(* IEC 61131-3 sources: Mizera_Tube/Plc (part 10) *)

LD   xEnFIR                        ** Abilita filtri FIR
ST   StPrFilterEnab                ** Stato precedente abilitazione filtri

LDN  xEnFIR                        ** Abilita filtri FIR
ST   EFCR_NF_DISABLE               ** NanoFIR subsystem disable

LDN  xEnFIR                        ** Abilita filtri FIR
ORN  EFSR_ACK_NF_DISABLE           ** ACK nanoFIR subsystem disable
AND  (
LD   xEnFIR                        ** Abilita filtri FIR
OR   EFSR_ACK_NF_DISABLE           ** ACK nanoFIR subsystem disable
)
ST   EFCR_SUBSYSTEM_EN             ** Filter subsystem master enable

LD   yLimiter                      ** Intervento limitatore
OR   xSetAlarm                     ** Forzamento allarme asse
*ANDN %ra0.28       ** Mem. collegamento richiesto con albero elettrico
ST   BAI_SETALARM                  ** ra0.27 Richiesta allarme asse

LD   xUnlock                       * reset gestax
R    yLimiter                      ** Intervento limitatore

LD   xEnFrComp                     ** Abilita friction compensation
ST   EFCR_FRICTION_COMP            ** Enable static friction comp.
ST   EFCR_RT_CHANGES_EN            ** Enable run-time changes (RT)

* Alarm if there is request of closeloop without drive enable

LD   BAI_CHAN                      ** ra0.0 Chiusura anello di posizione
AND  (
LD   %nvel11
EQ   3
OR   (
LD   %nvel11
EQ   4
)
)
ANDN BAI_AXEN                      ** Drive is enabled
ANDN LINK_SIMUL                    ** PLCFLAGS.16 LINK=SIMUL
ANDN AP_OPZIONI31                  ** pa3.31 Asse in simulato
ST   alarmEn                       ** Drive is disable, with enable request enabled

CAL  TON_ALARM_DISABLE (IN:=alarmEn,PT:=2000) ** Drive is disable, with enable request enabled

LD   TON_ALARM_DISABLE.Q
ST   yDriveNotEn                   ** Closeloop but drive not enabled (alarm)

LD  TON_ALARM_DISABLE.Q
JMPCN drive_is_enabled

LD   ALWAYS_ZERO                   ** PLCFLAGS.0  Flag sempre stato off
ST   AX_DRV_ENAB                   ** rg0.13 signal to understand all drives are enabled
drive_is_enabled:

* Comando bit avanti e indietro per i modi REF, JOG, INC

LD   CMD_START_AXIS                ** rgc0.5 Comando start assi canale
ANDN xLockRef                      ** Blocco avvio ciclo REF da canale
OR   xEnabRef                      ** Abilita avvio ciclo REF
AND  BCI_TAR                       ** rc0.8  Selettore modi operativi su REF (taratura)
AND  (
LDN  xZeroForced                   ** Forzamento asse tarato
ANDN BSC_SINGREF                   ** rgc0.18 Selezione modo REF singolo nel canale
OR   (
LD   xSelected                     ** Asse selezionato
AND  BSC_SINGREF                   ** rgc0.18 Selezione modo REF singolo nel canale
)
)
ST   StartRef                      ** Avvio ciclo di taratura

LD   CMD_PLUS_AXIS                 ** rgc0.0 Comando + assi canale
AND  xSelected                     ** Asse selezionato
OR   xJogPlus                      ** Comando manuale avanti
AND  AX_EXEC_MODE                  ** rgc0.3 Canale in JOG o INC
OR(
LD   StartRef                      ** Avvio ciclo di taratura
AND  AP_OPZIONI0                   ** pa3.0 Bit inversione direzione taratura
ANDN AsseNvel                      ** Asse di tipo NVEL
)
OR(
LD   StartRef                      ** Avvio ciclo di taratura
AND  NV_OPZIONI0                   ** pa1.0 Bit inversione direzione taratura (NVEL)
AND  AsseNvel                      ** Asse di tipo NVEL
)
ST   BAI_AV                        ** ra0.8 Comando avanti

LD   CMD_MINUS_AXIS                ** rgc0.1 Comando - assi canale
AND  xSelected                     ** Asse selezionato
OR   xJogMinus                     ** Comando manuale indietro
AND  AX_EXEC_MODE                  ** rgc0.3 Canale in JOG o INC
OR(
LD   StartRef                      ** Avvio ciclo di taratura
ANDN AP_OPZIONI0                   ** pa3.0 Bit inversione direzione taratura
ANDN AsseNvel                      ** Asse di tipo NVEL
)
OR(
LD   StartRef                      ** Avvio ciclo di taratura
ANDN NV_OPZIONI0                   ** pa1.0 Bit inversione direzione taratura (NVEL)
AND  AsseNvel                      ** Asse di tipo NVEL
)
ST   BAI_IND                       ** ra0.9 Comando indietro

* Passaggio finecorsa taratura e limite

LD   xRefLS                        ** Finecorsa di taratura
ST   BAI_FCRALL                    ** ra0.13 Finecorsa Taratura

LD   xPlusLS                       ** Finecorsa +
ST   BAI_FCHWAV                    ** ra0.10 Finecorsa avanti

LD   xMinusLS                      ** Finecorsa -
ST   BAI_FCHWIN                    ** ra0.11 Finecorsa indietro

* Reset asse in allarme

LD   CMD_RESET_AXIS                ** rgc0.4 Comando reset assi canale
ST   BAI_RESALARM                  ** ra0.15 Ripristino allarme asse

* Full-handshake motion block sul singolo asse

LD   BAO_STB_PLC_SYNC              ** ra22.16 strobe Full-handshake Motion block asse
AND  ACK_AX_FHMB                   ** rgc0.8 Abil. ACK Full-handshake Motion block per assi
ST   BAI_ACK_PLC_SYNC              ** ra0.26 ACK Full-handshake Motion block asse

* Taratura immediata (preset) sul singolo asse

LD   BSC_PRESETREF                 ** rgc0.19 Selezione modo REF preset nel canale
ST   BAI_TARAIM                    ** ra0.24 Selezione taratura immediata

LD   SC_QTAIMM                     ** rgc6 Quota per taratura immediata (preset)
ST   AI_QTAIMM                     ** ra2  Quota taratura immediata

* JOG DA VOLANTINO

LD   xSelected                     ** Asse selezionato
AND  PA_MOV_JOG                    ** rg0.8 Richiesta movim. da volantino in JOG
ST   JOG_AX.xax_ENABLE

LDN  JOG_AX.xax_ENABLE
ST   JOG_AX.xax_CLEAR

LD   JOG_AX.xax_ENABLE
AND  JOG_AX.yax_READY
ANDN JOG_AX.yax_RUNNING
AND  (
LDN  JOG_AX.yax_ENDERR
OR   JOG_AX.yax_ERRCODE.1
)
ST   JOG_AX.xax_START

LDN  PA_INV_DIR                    ** rg0.7 Movim. da volantino in direzione inversa
ST   JOG_AX.xax_REVERSE

CAL  JOG_AX

* Rileva il cambio di selezione asse

CAL  RT_AXSEL(CLK=xSelected)       ** Asse selezionato

LD   RT_AXSEL.Q                    ** Imp. selezione asse
S    AX_SEL_CHG                    ** rg0.12 Imp. modifica selezione asse

* POSIZIONAMENTO TRAMITE VOLANTINO

LD   xSelected                     ** Asse selezionato
ANDN RT_AXSEL.Q                    ** Imp. selezione asse
AND  PA_ENAB_POS                   ** rg0.9 Abilita posiz. asse da volantino
ST   POS_AX.xax_ENABLE

LDN  POS_AX.xax_ENABLE
ST   POS_AX.xax_CLEAR

LD   SG_QTAR_PAUX                  ** rg9 Quota Target per posiz. da puls. aux
NE   AO_QUOTA                      ** ra4  Quota asse
AND  POS_AX.xax_ENABLE
AND  POS_AX.yax_READY
ANDN POS_AX.yax_RUNNING
ANDN POS_AX.yax_ENDERR
ST   POS_AX.xax_START

LD   SG_QTAR_PAUX                  ** rg9 Quota Target per posiz. da puls. aux
ST   POS_AX.xax_QUOTA

LD   SG_VEL_PAUX                   ** rg14 Velocit� per posiz. da puls. aux
ST   POS_AX.xax_VEL

LD   SG_VEL_PAUX                   ** rg14 Velocit� per posiz. da puls. aux
GT   AP_VELMAX                     ** pa9 Velocit� massima
JMPCN END_VMAX

LD   AP_VELMAX                     ** pa9 Velocit� massima
ST   POS_AX.xax_VEL

END_VMAX:

CAL  POS_AX

* ALBERO ELETTRICO (per volantino e G4010)

LD   xSelected                     ** Asse selezionato
AND  PA_ENAB_ELS                   ** rg0.11 Abilita albero elettrico da volantino
OR   MemConnAE                     ** Mem. collegamento richiesto con albero elettrico
ANDN CAM_AX.yax_RUNNING
ST   EL_SH.xax_ENABLE

LDN  EL_SH.xax_ENABLE
OR   EL_SH.yax_ENDERR
ST   EL_SH.xax_CLEAR

LD   EL_SH.xax_ENABLE
AND  EL_SH.yax_READY
ANDN EL_SH.yax_ENDOK
ANDN EL_SH.yax_ENDERR
ANDN EL_SH.yax_RUNNING
ST   EL_SH.xax_START

LD   MemConnAE                     ** Mem. collegamento richiesto con albero elettrico
JMPC ELS_CON

LD   PA_INCJOG                     ** QPuls2 Quota incremento per posiz. da volantino
ST   EL_SH.xax_TRNUM

LD   EL_SH.xax_TRNUM
LT   1
JMPCN END_TRLIM

LD   1
ST   EL_SH.xax_TRNUM

END_TRLIM:

LD   1
ST   EL_SH.xax_TRDEN

LD   128
ST   EL_SH.xax_MODE

LD   SG_VOLAX                      ** rg16 Numero asse master per volantino
ST   EL_SH.xax_MASTER

JMP  ELS_END

ELS_CON:

LD   1
ST   EL_SH.xax_TRNUM
ST   EL_SH.xax_TRDEN

LD   0
ST   EL_SH.xax_MODE

LD   CONN_MAST                     ** rga1 Numero asse master per aggancio albero elettrico
ST   EL_SH.xax_MASTER

ELS_END:

CAL  EL_SH

* AX COUPLING

LD   MemConnCP                     ** Mem. collegamento richiesto con coupling
ANDN EL_SH.yax_RUNNING
ST   CAM_AX.xax_ENABLE

LDN  CAM_AX.xax_ENABLE
ST   CAM_AX.xax_CLEAR

LD   CAM_AX.xax_ENABLE
AND  CAM_AX.yax_READY
ANDN CAM_AX.yax_ENDOK
ANDN CAM_AX.yax_ENDERR
ST   CAM_AX.xax_START

LD   CP_TYPEC                      ** rga7 Tipo connessione per coupling
ST   CAM_AX.xax_MODE

*LD   0                      *non disponibile*
*ST   CAM_AX.xax_INSTANCE

LD   CP_MAST1                      ** rga3 Numero asse master 1 per coupling
ST   CAM_AX.xax_MASTER0

LD   CP_MAST2                      ** rga4 Numero asse master 2 per coupling
ST   CAM_AX.xax_MASTER1

LD   CP_MAST3                      ** rga5 Numero asse master 3 per coupling
ST   CAM_AX.xax_MASTER2

LD   CP_MAST4                      ** rga6 Numero asse master 4 per coupling
ST   CAM_AX.xax_MASTER3

LD   -1
ST   CAM_AX.xax_MASTER4

LD   -1
ST   CAM_AX.xax_MASTER5

CAL  CAM_AX

* Conferma comando effettuato

LD   MemConnAE                     ** Mem. collegamento richiesto con albero elettrico
AND  EL_SH.yax_RUNNING
AND  %ra8.14             * Conferma albero elettrico agganciato
OR   BAO_ALLM                      ** ra3.15  Asse in Allarme
OR   BAI_RESALARM                  ** ra0.15 Ripristino allarme asse
AND  REQ_CONN_AX                   ** rga0.0 Richiesta aggancio asse in albero elettrico
R    REQ_CONN_AX                   ** rga0.0 Richiesta aggancio asse in albero elettrico

LD   MemConnCP                     ** Mem. collegamento richiesto con coupling
AND  CAM_AX.yax_RUNNING
AND  %ra8.14             * Conferma albero elettrico agganciato
OR   BAO_ALLM                      ** ra3.15  Asse in Allarme
OR   BAI_RESALARM                  ** ra0.15 Ripristino allarme asse
AND  REQ_CONN_CP                   ** rga0.2 Richiesta aggancio asse in coupling
R    REQ_CONN_CP                   ** rga0.2 Richiesta aggancio asse in coupling

LDN  MemConnAE                     ** Mem. collegamento richiesto con albero elettrico
ANDN EL_SH.yax_RUNNING
ANDN MemConnCP                     ** Mem. collegamento richiesto con coupling
ANDN CAM_AX.yax_RUNNING
ANDN %ra8.14             * Conferma albero elettrico agganciato
OR   BAO_ALLM                      ** ra3.15  Asse in Allarme
OR   BAI_RESALARM                  ** ra0.15 Ripristino allarme asse
AND  REQ_SCON_AX                   ** rga0.1 Richiesta sgancio asse
R    REQ_SCON_AX                   ** rga0.1 Richiesta sgancio asse

LD   REQ_CONN_AX                   ** rga0.0 Richiesta aggancio asse in albero elettrico
OR   REQ_CONN_CP                   ** rga0.2 Richiesta aggancio asse in coupling
OR   REQ_SCON_AX                   ** rga0.1 Richiesta sgancio asse
S    BSY_CAX_PLC                   ** rg18.0 Busy aggancio/sgancio asse interno PLC

LD   MemConnAE                     ** Mem. collegamento richiesto con albero elettrico
AND  EL_SH.yax_RUNNING
AND  %ra8.14             * Conferma albero elettrico agganciato
ST   AX_CONN_OK                    ** rga2.0 Asse agganciato in albero elettrico

LD   MemConnCP                     ** Mem. collegamento richiesto con coupling
AND  CAM_AX.yax_RUNNING
AND  %ra8.14             * Conferma albero elettrico agganciato
ST   AX_CONCP_OK                   ** rga2.1 Asse agganciato in coupling

* Parallelo del segnale di allarme assi attivo

LD   BAO_ALLM                      ** ra3.15  Asse in Allarme
OR   BAO_ISO_ALARM                 ** ra19.4 Stato ALLARME all'interno del canale
S    CH_IN_ALARM                   ** rgc0.6 Asse in allarme nel canale

* Parallelo del segnale di asse in JOG presente

LD   BAO_ISO_JOG                   ** ra19.1 Stato JOG all'interno del canale
S    CH_AXJOG                      ** rgc0.21 Presente un asse in JOG nel canale

* Serie del segnale di assi tarati

LD   BAO_TARA                      ** ra3.14  Asse tarato
OR   xZeroForced                   ** Forzamento asse tarato
AND  CH_ZEROED                     ** rgc0.7 Assi tarati nel canale
ST   CH_ZEROED                     ** rgc0.7 Assi tarati nel canale

* Serie del segnale di assi fermi

LD   CH_STOPPED                    ** rgc0.9 Assi del canale fermi
AND  BAO_AFET                      ** ra3.0  Asse fermo teorico
ST   CH_STOPPED                    ** rgc0.9 Assi del canale fermi

* Registro asse selezionato per vis. cursore e quota asse

LD   xSelected                     ** Asse selezionato
JMPCN ENDAXSEL

LD   SG_AXNUM                      ** rg7 Numero asse all'interno del canale
ST   SG_AXSEL                      ** rg8 Asse selezionato per vis. cursore

LD   AO_QUOTA                      ** ra4  Quota asse
ST   SG_QACT_SEL                   ** rg10 Quota asse selezionato

LD   AsseNvel                      ** Asse di tipo NVEL
JMPC MinMaxNvel

LD   AP_MINQUOTA                   ** pa21 Quota minima
ST   SG_MINQ_SEL                   ** rg12 Quota minima asse selezionato

LD   AP_MAXQUOTA                   ** pa22 Quota massima
ST   SG_MAXQ_SEL                   ** rg13 Quota massima asse selezionato
JMP  ENDAXSEL

MinMaxNvel:
LD   NV_MINQUOTA                   ** pa10 Quota minima (NVEL)
ST   SG_MINQ_SEL                   ** rg12 Quota minima asse selezionato

LD   NV_MAXQUOTA                   ** pa11 Quota massima (NVEL)
ST   SG_MAXQ_SEL                   ** rg13 Quota massima asse selezionato

ENDAXSEL:

LD   xDisabVis                     ** Disabilita visualizzazone
JMPC DV

LD   SG_AXNUM                      ** rg7 Numero asse all'interno del canale
ADD  1
ST   SG_AXNUM                      ** rg7 Numero asse all'interno del canale

DV:

* Uscite di stato asse

LD   BAO_AFET                      ** ra3.0  Asse fermo teorico
ST   yStopped                      ** Asse fermo

LD   BAO_AXAV                      ** ra3.2  Direzione moto asse avanti
ST   yForward                      ** Direzione asse avanti

* Il mantenimento dell'uscita di abilitazione azionamento
* al rilascio del JOG OPEN su un asse con freno ha effetto
* solo se l'uscita � comandata dal PLC, in caso contrario
* on motore e freno si disattivano insieme, e su un asse
* verticale questo potrebbe determinare una caduta.
* Aggiunto TOF_ONMOT per evitare l'errore saltuario
* "Richiesta allarme I/O di controllo"

CAL TOF_ONMOT(IN=BAO_ONMT, PT=150) ** ra3.10  Richiesta abilitazione azionamento

LD   TOF_FRENO.Q                   ** Fine tempo chiusura freno
AND  ST_JOGOPEN                    ** rgc0.17 Stato JOG OPEN attivo
AND  xBrakeEnab                    ** Abilita gestione freno (provv.)
OR   TOF_ONMOT.Q                   ** Fine tempo on motore
ST   yClosedLoop                   ** Asse in coppia

LD   BAO_ORDM                      ** ra3.13  Ordine di moto
ST   yOrdineMoto                   ** Ordine di moto asse

LD   BAO_TARA                      ** ra3.14  Asse tarato
OR   xZeroForced                   ** Forzamento asse tarato
ST   yZeroed                       ** Asse tarato

LD   BAO_ALLM                      ** ra3.15  Asse in Allarme
OR (
LD   REQ_CONN_AX                   ** rga0.0 Richiesta aggancio asse in albero elettrico
OR   REQ_CONN_CP                   ** rga0.2 Richiesta aggancio asse in coupling
OR   REQ_SCON_AX                   ** rga0.1 Richiesta sgancio asse
ANDN RichCloseLoop                 ** Richiesta di messa in coppia
)
ST   yInAlarm                      ** Asse in allarme

END_FUNCTION_BLOCK

* FB DECODIFICA SELEZIONE ASSE

VAR_IN_OUT
CC_REGS AT %cc;
END_VAR

FUNCTION_BLOCK DEC_SEL_ASSE

VAR_INPUT
xMaskAxSel: DWORD; * Maschera compressa asse selezionato
END_VAR

VAR_OUTPUT
yExtMask: DWORD; * Maschera estesa asse selezionato
yNumAsse: DWORD; * Numero system-wide asse selezionato
END_VAR

VAR
MaskCnf: DWORD; * Maschera estesa assi configurati
MaskSel: DWORD; * Maschera compressa asse selezionato
Index: DWORD; * Indice registro numero system-wide asse
END_VAR

LD   1
ST   yExtMask                      ** Maschera estesa asse selezionato

LD   2
ST   Index                         ** Indice registro numero system-wide asse

LD   xMaskAxSel                    ** Maschera compressa asse selezionato
ST   MaskSel                       ** Maschera compressa asse selezionato

LD   CC_MASKAXES                   ** cc1 Maschera configurazione assi nel canale
ANDN %DisabVisAX
ST   MaskCnf                       ** Maschera estesa assi configurati

LOOP:

LDN  MaskCnf.0
JMPC NEXT_CNF

LD   MaskSel.0
JMPC END_LOOP

LD   MaskSel                       ** Maschera compressa asse selezionato
SHR  1
ST   MaskSel                       ** Maschera compressa asse selezionato

NEXT_CNF:

LD   MaskCnf                       ** Maschera estesa assi configurati
SHR  1
ST   MaskCnf                       ** Maschera estesa assi configurati

LD   MaskCnf                       ** Maschera estesa assi configurati
EQ   0
OR   (
LD   MaskSel                       ** Maschera compressa asse selezionato
EQ   0
)
JMPC MASK_NULL

LD   yExtMask                      ** Maschera estesa asse selezionato
SHL  1
ST   yExtMask                      ** Maschera estesa asse selezionato

LD   Index                         ** Indice registro numero system-wide asse
ADD  1
ST   Index                         ** Indice registro numero system-wide asse

JMP  LOOP

MASK_NULL:

LD   0
ST   yExtMask                      ** Maschera estesa asse selezionato

LD   -1
ST   yNumAsse                      ** Numero system-wide asse selezionato

JMP  END_SEL

END_LOOP:

LD   CC_REGS[Index]                ** Indice registro numero system-wide asse
ST   yNumAsse                      ** Numero system-wide asse selezionato

END_SEL:

END_FUNCTION_BLOCK

* FB TOGGLE, per ora non usato

FUNCTION_BLOCK TOGGLE

VAR_INPUT
CLK: BOOL; * Input toggle
R: BOOL; * Reset forzato
END_VAR

VAR_OUTPUT
Q: BOOL; * Output toggle
END_VAR

VAR
PrevStatus: BOOL; * Stato precedente input toggle
SetActive:  BOOL; * Impulso attivazione toggle
Status: BOOL; * Stato interno toggle
END_VAR

LD   CLK                           ** Input toggle
ANDN PrevStatus                    ** Stato precedente input toggle
ANDN Status                        ** Stato interno toggle
S    Status                        ** Stato interno toggle
ST   SetActive                     ** Impulso attivazione toggle

LD   CLK                           ** Input toggle
ANDN PrevStatus                    ** Stato precedente input toggle
ANDN SetActive                     ** Impulso attivazione toggle
OR   R                             ** Reset forzato
R    Status                        ** Reset forzato

LD   CLK                           ** Input toggle
ST   PrevStatus                    ** Stato precedente input toggle

LD   Status                        ** Stato interno toggle
ST   Q                             ** Output toggle

END_FUNCTION_BLOCK

* FB GESTIONE CAMBIO UTENSILE CON ASSE ROUND TABLE

FUNCTION_BLOCK GESTTABLE

VAR_INPUT
xSelected: BOOL; * Asse selezionato
xEnabOp: BOOL; * Sicurezze rotazione asse
xSelCSingRot: BOOL; * Selezione rotazione ciclo singolo
END_VAR

VAR_OUTPUT
yWaitMFun: BOOL; * Ritarda ACK funzioni M
yToolChangeRun: BOOL; * Cambio utensile in corso
yAlmPos: BOOL;  * Errore posizione finale
END_VAR

VAR
#defcom R_TRIG1.Q Fronte per cambio utensile da programma (M6)
#defcom R_TRIG2.Q Fronte per ciclo continuo singolo

R_TRIG1: R_TRIG;
R_TRIG2: R_TRIG;

RTABLE: AX_RTABLE;

Appoggio:       BOOL; * Appoggio
ChToolRun:      BOOL; * Cambio utensile in corso
CmdCicSing:     BOOL; * Comando ciclo singolo rotazione attivo
ToolFromPP:     DWORD; * Utensile richiesto da part program
END_VAR

* Condizioni per cambio utensile da programma (M6)

LD   FUN_M6                        ** rgc1.6  Funzione M6 attiva
AND  xEnabOp                       ** Sicurezze rotazione asse
ANDN ChToolRun                     ** Cambio utensile in corso
ST   Appoggio                      ** Appoggio

CAL  R_TRIG1(CLK=Appoggio)         ** Appoggio

* Campiona funzione T solo sulla M6

LDN  R_TRIG1.Q                     ** Fronte per cambio utensile da programma (M6)
JMPC ENDTOOLPP

LD   CO_TFUN                       ** rc11 Registro funzioni T
ST   ToolFromPP                    ** Utensile richiesto da part program

ENDTOOLPP:

* Condizioni per ciclo continuo singolo

LD   CMD_MINUS_AXIS                ** rgc0.1 Comando - assi canale
OR   CMD_PLUS_AXIS                 ** rgc0.0 Comando + assi canale
OR   CMD_START_AXIS                ** rgc0.5 Comando start assi canale
AND  xSelCSingRot                  ** Selezione rotazione ciclo singolo
AND  xSelected                     ** Asse selezionato
AND  xEnabOp                       ** Sicurezze rotazione asse
ANDN yAlmPos                       ** Errore posizione finale
ST   CmdCicSing                    ** Comando ciclo singolo rotazione attivo

CAL  R_TRIG2(CLK=CmdCicSing)       ** Comando ciclo singolo rotazione attivo

* Ciclo cambio utensile

LD   R_TRIG1.Q                     ** Fronte per cambio utensile da programma (M6)
OR   R_TRIG2.Q                     ** Fronte per ciclo continuo singolo
S    ChToolRun                     ** Cambio utensile in corso

LD   RTABLE.yax_ENDOK
OR   CMD_RESET_AXIS                ** rgc0.4 Comando reset assi canale
OR   BCI_MAN                       ** rc0.9  Selettore modi operativi su JOG (manuale)
OR   BCI_TAR                       ** rc0.8  Selettore modi operativi su REF (taratura)
R    ChToolRun                     ** Cambio utensile in corso

LD   ChToolRun                     ** Cambio utensile in corso
ST   yToolChangeRun                ** Cambio utensile in corso

* Comando per arresto STEP asse con rilascio pulsante

LDN  CMD_RESET_AXIS                ** rgc0.4 Comando reset assi canale
AND  BCO_CANREADY                  ** rc8.2  Canale Ready
AND  (
LD   CmdCicSing                    ** Comando ciclo singolo rotazione attivo
ORN  xSelCSingRot                  ** Selezione rotazione ciclo singolo
ORN  RTABLE.yax_RUNNING
)
ST   RTABLE.xax_ENABLE

LD   CmdCicSing                    ** Comando ciclo singolo rotazione attivo
ORN  xSelCSingRot                  ** Selezione rotazione ciclo singolo
AND  ChToolRun                     ** Cambio utensile in corso
AND  RTABLE.yax_READY
ANDN RTABLE.yax_ENDOK
ANDN RTABLE.yax_ENDERR
ST   RTABLE.xax_START

LDN  ChToolRun                     ** Cambio utensile in corso
AND  RTABLE.yax_ENDOK
OR   (
LD   RTABLE.yax_ERRCODE.1
AND  xSelCSingRot                  ** Selezione rotazione ciclo singolo
)
OR   CMD_RESET_AXIS                ** rgc0.4 Comando reset assi canale
ST   RTABLE.xax_CLEAR

LD   xSelCSingRot                  ** Selezione rotazione ciclo singolo
ANDN CMD_START_AXIS                ** rgc0.5 Comando start assi canale
ST   RTABLE.xax_POSMODE

LD   CMD_PLUS_AXIS                 ** rgc0.0 Comando + assi canale
OR   CMD_MINUS_AXIS                ** rgc0.1 Comando - assi canale
ST   RTABLE.xax_INCMODE

LD   CMD_MINUS_AXIS                ** rgc0.1 Comando - assi canale
ST   RTABLE.xax_REVERSE

LD   xSelCSingRot                  ** Selezione rotazione ciclo singolo
JMPC DATI_ROTSING

LD   ToolFromPP                    ** Utensile richiesto da part program
ST   RTABLE.xax_QUOTA

LD   AP_VELMAX                     ** pa9 Velocit� massima
ST   RTABLE.xax_VEL

JMP  END_DATI_ROTSING

DATI_ROTSING:

LD   1
ST   RTABLE.xax_QUOTA

LD   AP_VELMAN                     ** pa23 Velocit� di JOG
ST   RTABLE.xax_VEL

LD   CI_FIXINCR                    ** rc4  Quota per incrementi fissi
EQ   0
JMPC END_DATI_ROTSING

LD   CI_FIXINCR                    ** rc4  Quota per incrementi fissi
DIV  1000          ** diviso 1000
ST   RTABLE.xax_QUOTA

END_DATI_ROTSING:

CAL  RTABLE

LDN  RTABLE.yax_ERRCODE.1
ORN  xSelCSingRot                  ** Selezione rotazione ciclo singolo
AND  RTABLE.yax_ENDERR
ST   yAlmPos                       ** Errore posizione finale

* Ritarda ACK M da cambio utensile

LD   ChToolRun                     ** Cambio utensile in corso
AND  FUN_M6                        ** rgc1.6  Funzione M6 attiva
ST   yWaitMFun                     ** Ritarda ACK funzioni M

END_FUNCTION_BLOCK

* --------------------------------------------*
* Blocco Funzionale ciclo di taratura completo
* --------------------------------------------*

FUNCTION_BLOCK CYC_HOMING

VAR_INPUT
xax_ENABLE:   BOOL;       * abilita FB
xax_START:    BOOL;       * start richiesta azione
xax_CLEAR:    BOOL;       * conferma fine comando
xax_IMMDATA:  BOOL;       * dati (vmax, rampe) immediati
                          * 0 = carica dati di sistema
                          * 1 = carica dati da input FB
xax_REVERSE:  BOOL;       * 0 = quote decrescenti, 1 = quote crescenti
xax_MODE:     DWORD;      * Modo di taratura
xax_QUOTA:    DWORD;      * Quota di taratura ( 0.001 mm )
xax_VELFC:    DWORD;      * Velocita' ricerca micro ( mm/min )
xax_VEL:      DWORD;      * Velocita' ricerca tacca ( mm/min )
xax_VMAX:     DWORD;      * Velocita' massima ( mm/min )
xax_ACCEL:    DWORD;      * Accelerazione e decelerazione (msec o mm/s2)

END_VAR

VAR_OUTPUT
yax_READY:    BOOL;       * FB pronto per START
yax_RUNNING:  BOOL;       * Esecuzione FB in corso
yax_ENDOK:    BOOL;       * Comando terminato correttamente
yax_ENDERR:   BOOL;       * Comando terminato non correttamente
yax_ERRCODE:  DWORD;      * codice errore ( maschera bit )
END_VAR

VAR
TarQuota: DWORD; * Quota di taratura
VelMic: DWORD; * Velocita' ricerca micro
VelTac: DWORD; * Velocita' ricerca tacca
VelMax: DWORD; * Velocita' massima
AccDec: DWORD; * Accelerazione e decelerazione
TarMode: DWORD; * Modo di taratura
DirZero: BOOL; * Direzione ric. zero: 0 = quote decrescenti, 1 = quote crescenti

ZCOn: BOOL; * Ciclo ricerca zero attivo
ZCRicAttMicro: BOOL; * Ciclo ricerca zero: ricerca attivazione micro
ZCRicRilMicro: BOOL; * Ciclo ricerca zero: ricerca rilascio micro
ZCRicTacca: BOOL; * Ciclo ricerca zero: ricerca tacca
ZCEnabLSW: BOOL; * Ciclo ricerca zero: riabilita limiti SW
ZCPark: BOOL; * Ciclo ricerca zero: parcheggio
ZCEndOK: BOOL; * Ciclo ricerca zero terminato OK
ZCEndErr: BOOL; * Ciclo ricerca zero terminato con errore

Appoggio: BOOL; * Variabile di appoggio
NoUseMicro: BOOL; * Ciclo senza fase di ricerca micro
TaraFC: BOOL; * Ciclo zero su finecorsa (senza tacca)
EnabPark: BOOL; * Ciclo con parcheggio finale

HOMFB: AX_HOMING;
JOGFB: AX_JOGGING;
POSFB: AX_POSIZ;
CNTFB: AX_CONTROLS;
END_VAR

LD   xax_IMMDATA                   ** dati (vmax, rampe) immediati
JMPC IMMDATA

LD   AP_AXTYPE                     ** pa0 Tipo asse
EQ   20
JMPC NV_DATA

LD   AP_TARQUOTA                   ** pa18 Quota di taratura
ST   TarQuota                      ** Quota di taratura

LD   AP_VELMICRO                   ** pa19 Velocit� ricerca micro in taratura
ST   VelMic                        ** Velocita' ricerca micro

LD   AP_VELTACCA                   ** pa20 Velocit� ricerca tacca in taratura
ST   VelTac                        ** Velocita' ricerca tacca

LD   AP_VELMAX                     ** pa9 Velocit� massima
ST   VelMax                        ** Velocita' massima

LD   AP_ACCEL                      ** pa1 Accelerazione massima
ST   AccDec                        ** Accelerazione e decelerazione

LD   AP_TARTYPE                    ** pa16 Tipo di taratura
ST   TarMode                       ** Modo di taratura

LD   AP_OPZIONI0                   ** pa3.0 Bit inversione direzione taratura
ST   DirZero                       ** Direzione ric. zero: 0 = quote decrescenti, 1 = quote crescenti

JMP  END_DATA

NV_DATA:

LD   NV_TARQUOTA                   ** pa7 Quota di taratura (NVEL)
ST   TarQuota                      ** Quota di taratura

LD   NV_VELMICRO                   ** pa8 Velocit� ricerca micro in taratura (NVEL)
ST   VelMic                        ** Velocita' ricerca micro

LD   NV_VELTACCA                   ** pa9 Velocit� ricerca tacca in taratura (NVEL)
ST   VelTac                        ** Velocita' ricerca tacca

LD   NV_VELMAX                     ** pa4 Velocit� massima (NVEL)
ST   VelMax                        ** Velocita' massima

LD   0
ST   AccDec                        ** Accelerazione e decelerazione

LD   NV_TARTYPE                    ** pa6 Tipo di taratura (NVEL)
ST   TarMode                       ** Modo di taratura

LD   NV_OPZIONI0                   ** pa1.0 Bit inversione direzione taratura (NVEL)
ST   DirZero                       ** Direzione ric. zero: 0 = quote decrescenti, 1 = quote crescenti

JMP  END_DATA

IMMDATA:

LD   xax_QUOTA                     ** Quota di taratura ( 0.001 mm )
ST   TarQuota                      ** Quota di taratura

LD   xax_VELFC                     ** Velocita' ricerca micro ( mm/min )
ST   VelMic                        ** Velocita' ricerca micro

LD   xax_VEL                       ** Velocita' ricerca tacca ( mm/min )
ST   VelTac                        ** Velocita' ricerca tacca

LD   xax_VMAX                      ** Velocita' massima ( mm/min )
ST   VelMax                        ** Velocita' massima

LD   xax_ACCEL                     ** Accelerazione e decelerazione (msec o mm/s2)
ST   AccDec                        ** Accelerazione e decelerazione

LD   xax_MODE                      ** Modo di taratura
ST   TarMode                       ** Modo di taratura

LD   xax_REVERSE                   ** 0 = quote decrescenti, 1 = quote crescenti
ST   DirZero                       ** Direzione ric. zero: 0 = quote decrescenti, 1 = quote crescenti

END_DATA:

LD   AP_DRVTYPE                    ** nvel11 Tipo drive (0=analogico)
NE   0
OR   (
LD   TarMode                       ** Modo di taratura
EQ   2
)
ST   NoUseMicro                    ** Ciclo senza fase di ricerca micro

LD   TarMode                       ** Modo di taratura
EQ   3
OR   (
LD   TarMode                       ** Modo di taratura
EQ   4
)
ANDN NoUseMicro                    ** Ciclo senza fase di ricerca micro
ST   TaraFC                        ** Ciclo zero su finecorsa (senza tacca)

LD   TarMode                       ** Modo di taratura
EQ   1
OR   (
LD   TarMode                       ** Modo di taratura
EQ   4
)
ANDN NoUseMicro                    ** Ciclo senza fase di ricerca micro
ST   EnabPark                      ** Ciclo con parcheggio finale

LD   xax_START                     ** start richiesta azione
S    ZCOn                          ** Ciclo ricerca zero attivo

LD   CNTFB.yax_ENDOK
OR   NoUseMicro                    ** Ciclo senza fase di ricerca micro
AND  ZCOn                          ** Ciclo ricerca zero attivo
S    ZCRicAttMicro                 ** Ciclo ricerca zero: ricerca attivazione micro

LD   BAI_FCRALL                    ** ra0.13 Finecorsa Taratura
OR   NoUseMicro                    ** Ciclo senza fase di ricerca micro
AND  ZCRicAttMicro                 ** Ciclo ricerca zero: ricerca attivazione micro
S    ZCRicRilMicro                 ** Ciclo ricerca zero: ricerca rilascio micro

LDN  BAI_FCRALL                    ** ra0.13 Finecorsa Taratura
OR   NoUseMicro                    ** Ciclo senza fase di ricerca micro
AND  ZCRicRilMicro                 ** Ciclo ricerca zero: ricerca rilascio micro
S    ZCRicTacca                    ** Ciclo ricerca zero: ricerca tacca

LD   HOMFB.yax_ENDOK
AND  ZCRicTacca                    ** Ciclo ricerca zero: ricerca tacca
S    ZCEnabLSW                     ** Ciclo ricerca zero: riabilita limiti SW

LD   CNTFB.yax_ENDOK
AND  ZCEnabLSW                     ** Ciclo ricerca zero: riabilita limiti SW
S    ZCPark                        ** Ciclo ricerca zero: parcheggio

LD   POSFB.yax_ENDOK
ORN  EnabPark                      ** Ciclo con parcheggio finale
AND  ZCPark                        ** Ciclo ricerca zero: parcheggio
S    ZCEndOK                       ** Ciclo ricerca zero terminato OK

LDN  xax_ENABLE                    ** abilita FB
AND  ZCOn                          ** Ciclo ricerca zero attivo
S    ZCEndErr                      ** Ciclo ricerca zero terminato con errore

LD   ZCEndOK                       ** Ciclo ricerca zero terminato OK
OR   ZCEndErr                      ** Ciclo ricerca zero terminato con errore
AND  xax_CLEAR                     ** conferma fine comando
R    ZCOn                          ** Ciclo ricerca zero attivo
R    ZCRicAttMicro                 ** Ciclo ricerca zero: ricerca attivazione micro
R    ZCRicRilMicro                 ** Ciclo ricerca zero: ricerca rilascio micro
R    ZCRicTacca                    ** Ciclo ricerca zero: ricerca tacca
R    ZCEnabLSW                     ** Ciclo ricerca zero: riabilita limiti SW
R    ZCPark                        ** Ciclo ricerca zero: parcheggio
R    ZCEndOK                       ** Ciclo ricerca zero terminato OK
R    ZCEndErr                      ** Ciclo ricerca zero terminato con errore

* Movimento asse in JOG

LDN  ZCRicTacca                    ** Ciclo ricerca zero: ricerca tacca
ORN  JOGFB.yax_RUNNING
AND  xax_ENABLE                    ** abilita FB
ST   JOGFB.xax_ENABLE

LD   ZCRicAttMicro                 ** Ciclo ricerca zero: ricerca attivazione micro
ANDN ZCRicTacca                    ** Ciclo ricerca zero: ricerca tacca
ST   Appoggio                      ** Variabile di appoggio

LD   xax_CLEAR                     ** conferma fine comando
AND  JOGFB.yax_ENDERR
ORN  Appoggio                      ** Variabile di appoggio
ST   JOGFB.xax_CLEAR

LD   Appoggio                      ** Variabile di appoggio
AND  JOGFB.xax_ENABLE
AND  JOGFB.yax_READY
ANDN JOGFB.yax_ENDOK
ANDN JOGFB.yax_ENDERR
ST   JOGFB.xax_START

LD   ALWAYS_ONE                    ** PLCFLAGS.1  Flag sempre stato on
ST   JOGFB.xax_VARVEL

*LD   DirZero
*ST   JOGFB.xax_REVERSE

LD   ZCRicRilMicro                 ** Ciclo ricerca zero: ricerca rilascio micro
JMPC RILMICRO

LD   VelMic                        ** Velocita' ricerca micro
ST   JOGFB.xax_VEL

JMP  END_VJOG

RILMICRO:

LD   VelTac                        ** Velocita' ricerca tacca
ST   JOGFB.xax_VEL

END_VJOG:

LD   DirZero                       ** Direzione ric. zero: 0 = quote decrescenti, 1 = quote crescenti
AND  ZCRicRilMicro                 ** Ciclo ricerca zero: ricerca rilascio micro
OR   (
LDN  DirZero                       ** Direzione ric. zero: 0 = quote decrescenti, 1 = quote crescenti
ANDN ZCRicRilMicro                 ** Ciclo ricerca zero: ricerca rilascio micro
)
JMPCN REV_VEL_JOG

LD   JOGFB.xax_VEL
MUL  -1
ST   JOGFB.xax_VEL

REV_VEL_JOG:

CAL  JOGFB

* Chiamata FB standard ricerca tacca (per assi analogici),
* che per gli assi digitali realizza l'intero ciclo di zero.

LD   xax_ENABLE                    ** abilita FB
ST   HOMFB.xax_ENABLE

LD   ZCRicTacca                    ** Ciclo ricerca zero: ricerca tacca
ANDN ZCEnabLSW                     ** Ciclo ricerca zero: riabilita limiti SW
ST   Appoggio                      ** Variabile di appoggio

LD   xax_CLEAR                     ** conferma fine comando
AND  HOMFB.yax_ENDERR
ORN  Appoggio                      ** Variabile di appoggio
ST   HOMFB.xax_CLEAR

LD   Appoggio                      ** Variabile di appoggio
ANDN JOGFB.yax_RUNNING
AND  HOMFB.xax_ENABLE
AND  HOMFB.yax_READY
ANDN HOMFB.yax_ENDOK
ANDN HOMFB.yax_ENDERR
ST   HOMFB.xax_START

LD   ALWAYS_ONE                    ** PLCFLAGS.1  Flag sempre stato on
ST   HOMFB.xax_IMMDATA

LDN  DirZero                       ** Direzione ric. zero: 0 = quote decrescenti, 1 = quote crescenti
ST   HOMFB.xax_REVERSE

LD   TarMode                       ** Modo di taratura
ST   HOMFB.xax_MODE

LD   TaraFC                        ** Ciclo zero su finecorsa (senza tacca)
JMPCN FORCE_IMM

LD   2
ST   HOMFB.xax_MODE

FORCE_IMM:

LD   TarQuota                      ** Quota di taratura
ST   HOMFB.xax_QUOTA

LD   VelTac                        ** Velocita' ricerca tacca
ST   HOMFB.xax_VEL

LD   VelMax                        ** Velocita' massima
ST   HOMFB.xax_VMAX

LD   AccDec                        ** Accelerazione e decelerazione
ST   HOMFB.xax_ACCEL

CAL  HOMFB

* Posizionamento asse a quota di parcheggio

LD   xax_ENABLE                    ** abilita FB
ST   POSFB.xax_ENABLE

LD   ZCPark                        ** Ciclo ricerca zero: parcheggio
ANDN ZCEndOK                       ** Ciclo ricerca zero terminato OK
ST   Appoggio                      ** Variabile di appoggio

LD   xax_CLEAR                     ** conferma fine comando
AND  POSFB.yax_ENDERR
ORN  Appoggio                      ** Variabile di appoggio
ST   POSFB.xax_CLEAR

LD   Appoggio                      ** Variabile di appoggio
AND  POSFB.xax_ENABLE
AND  POSFB.yax_READY
ANDN POSFB.yax_ENDOK
ANDN POSFB.yax_ENDERR
ST   POSFB.xax_START

LD   AP_PARKQTA                    ** pa31 Quota di parcheggio
ST   POSFB.xax_QUOTA

LD   AP_VELMAX                     ** pa9 Velocit� massima
ST   POSFB.xax_VEL

CAL  POSFB

* Disabilitazione bit asse tarato, per evitare che il JOG
* si fermi sul limite SW, e successiva riabilitazione

LD   xax_ENABLE                    ** abilita FB
ST   CNTFB.xax_ENABLE

LD   ZCOn                          ** Ciclo ricerca zero attivo
ANDN ZCRicAttMicro                 ** Ciclo ricerca zero: ricerca attivazione micro
OR   (
LD   ZCEnabLSW                     ** Ciclo ricerca zero: riabilita limiti SW
ANDN ZCPark                        ** Ciclo ricerca zero: parcheggio
)
ST   Appoggio                      ** Variabile di appoggio

LD   xax_CLEAR                     ** conferma fine comando
AND  CNTFB.yax_ENDERR
ORN  Appoggio                      ** Variabile di appoggio
ST   CNTFB.xax_CLEAR

LD   Appoggio                      ** Variabile di appoggio
AND  CNTFB.xax_ENABLE
AND  CNTFB.yax_READY
ANDN CNTFB.yax_ENDOK
ANDN CNTFB.yax_ENDERR
ST   CNTFB.xax_START

LD   ZCRicTacca                    ** Ciclo ricerca zero: ricerca tacca
JMPC RIAB_LIMSW

LD   16#28
ST   CNTFB.xax_DISMASK

LD   0
ST   CNTFB.xax_ENMASK

JMP  END_LIMSW

RIAB_LIMSW:

LD   0
ST   CNTFB.xax_DISMASK

LD   16#8
ST   CNTFB.xax_ENMASK

END_LIMSW:

CAL  CNTFB

* Comando uscite

LD   ZCOn                          ** Ciclo ricerca zero attivo
ANDN ZCEndOK                       ** Ciclo ricerca zero terminato OK
ST   yax_RUNNING                   ** Esecuzione FB in corso

LD   HOMFB.yax_READY
AND  JOGFB.yax_READY
AND  POSFB.yax_READY
AND  CNTFB.yax_READY
ANDN yax_RUNNING                   ** Esecuzione FB in corso
ST   yax_READY                     ** FB pronto per START

LD   ZCEndOK                       ** Ciclo ricerca zero terminato OK
ST   yax_ENDOK                     ** Comando terminato correttamente

LD   JOGFB.yax_ENDERR
ANDN ZCRicTacca                    ** Ciclo ricerca zero: ricerca tacca
OR   HOMFB.yax_ENDERR
OR   POSFB.yax_ENDERR
OR   CNTFB.yax_ENDERR
OR   ZCEndErr                      ** Ciclo ricerca zero terminato con errore
ST   yax_ENDERR                    ** Comando terminato non correttamente

LD   ZCEndErr                      ** Ciclo ricerca zero terminato con errore
JMPCN GEN_ERR

LD   2
ST   yax_ERRCODE                   ** codice errore ( maschera bit )

GEN_ERR:

LD   JOGFB.yax_ERRCODE
ST   yax_ERRCODE                   ** codice errore ( maschera bit )

LD   HOMFB.yax_ENDERR
JMPCN HOMERR

LD   HOMFB.yax_ERRCODE
ST   yax_ERRCODE                   ** codice errore ( maschera bit )

HOMERR:

LD   POSFB.yax_ENDERR
JMPCN POSERR

LD   POSFB.yax_ERRCODE
ST   yax_ERRCODE                   ** codice errore ( maschera bit )

POSERR:

LD   CNTFB.yax_ENDERR
JMPCN CNTERR

LD   CNTFB.yax_ERRCODE
ST   yax_ERRCODE                   ** codice errore ( maschera bit )

CNTERR:

END_FUNCTION_BLOCK

VAR_IN_OUT
QTA_TARA_SLAVE AT %pa18; * pa18 Quota di taratura asse
END_VAR

* FB GESTIONE ASSI GANTRY

FUNCTION_BLOCK GST_GANTRY

VAR_INPUT
xRefCycle: BOOL; * Comando esecuzione ciclo di taratura
xReqPreset: BOOL; * Richiesta preset slave alla quota del master
xReqAllin: BOOL; * Richiesta allineamento slave alla quota del master
xReqSgancio: BOOL; * Richiesta sgancio gantry
xReqAggancio: BOOL; * Richiesta aggancio gantry
xReset: BOOL; * Reset comandi gantry
xLSZeroM: BOOL; * Finecorsa taratura asse master
xLSZeroS: BOOL; * Finecorsa taratura asse slave
xExtCmd: BOOL; * Selezione comandi REF-JOG esterni (da canale)
xParkCycle: BOOL; * Abilita ciclo parcheggio a fine taratura
xZeroSetup: BOOL; * Esclude allineamento a fine taratura
xNoAlarm: BOOL; * Esclude allarme massimo disallineamento
xAuxBusy: BOOL; * Canale ausiliario impegnato
xEmer: BOOL; * Condizioni di emergenza che forzano l'apertura del gantry
xAutZeroSetup: BOOL; * Modifica automatica quota taratura a fine setup
xNMaster: DWORD; * Numero asse master
xNSlave: DWORD; * Numero asse slave
xParkSpeed: DWORD; * Velocit� di parcheggio
END_VAR

VAR_OUTPUT
yGantryOff: BOOL; * Accoppiamento gantry non attivo
yGantryOn: BOOL; * Accoppiamento gantry attivo
yEndCycRef: BOOL; * Fine ciclo taratura gantry
yEndPrAll: BOOL; * Fine preset o allineamento slave a quota master
yGrant: BOOL; * Richiesta comando assi da PLC
yRefM: BOOL; * Richiesta ciclo zero su asse master
yRefS: BOOL; * Richiesta ciclo zero su asse slave
yOnOff: BOOL; * Comando aggancio-sgancio in corso
yAlPr: BOOL; * Comando allineamento-preset dopo ripristino emergenza in corso
yRefAlarm: BOOL; * Allarme allineamento durante ciclo zero
yPresetReq: BOOL; * Richesta preset asse Slave
ycn_ERRCODE: DWORD; *  Function-Block error code
END_VAR

VAR
GantryOnS: BOOL; * Gantry attivo su asse slave
AlarmS: BOOL; * Allarme su asse slave
AxFermoS: BOOL; * Asse slave fermo
AxTaratoS: BOOL; * Asse slave tarato
IsoNullS: BOOL; * Asse slave in ISO nullo
Ref1LS: BOOL; * Ciclo taratura con 1 finecorsa
MemZeroM: BOOL; * Mem. asse master tarato
EndZeroM: BOOL; * Ciclo taratura asse master effettuato
MemZeroS: BOOL; * Mem. asse slave tarato
EndZeroS: BOOL; * Ciclo taratura asse slave effettuato
CTGPreset: BOOL; * Ciclo tara gantry: preset iniziale
CTGFirstAgg: BOOL; * Ciclo tara gantry: primo aggancio gantry
CTGZeroM: BOOL; * Ciclo tara gantry: ricerca zero su asse master
CTGSlaveAgg: BOOL; * Ciclo tara gantry: aggancio gantry slave-master
CTGZeroS: BOOL; * Ciclo tara gantry: ricerca zero su asse slave
CTGLastSga: BOOL; * Ciclo tara gantry: ultimo sgancio gantry
CTGAllin: BOOL; * Ciclo tara gantry: posiziona slave alla quota master
CTGLastAgg: BOOL; * Ciclo tara gantry: ultimo aggancio gantry
CTGPark: BOOL; * Ciclo tara gantry: parcheggio gantry
CPASga: BOOL; * Ciclo allinea gantry: sgancio gantry
CPAExec: BOOL; * Ciclo allinea gantry: esegue preset o allineamento
CPARiagg: BOOL; * Ciclo allinea gantry: riaggancio gantry
CARSga: BOOL; * Ciclo allinea al ripristino emergenza: sgancio gantry
CARAllin: BOOL; * Ciclo allinea al ripristino emergenza: esegue allineamento
CARRiagg: BOOL; * Ciclo allinea al ripristino emergenza: riaggancio gantry
ForzAggancio: BOOL; * Cond. forzamento aggancio gantry (anche se lo � gi�)
CodeLibereSlave: BOOL; * Nessun comando su coda slave
MemAggancio: BOOL; * Mem. aggancio gantry
MemSetupDone: BOOL; * Mem. eseguito ciclo setup
AllDopoEmer: BOOL; * Abilita allineamento gantry dopo emergenza
Appoggio: BOOL; * Appoggio
PosMaster: DWORD; * Quota attuale asse master
PosSlave: DWORD; * Quota attuale asse slave

#defcom RT_TARAM.Q Imp. asse master tarato
RT_TARAM: R_TRIG;
#defcom RT_TARAS.Q Imp. asse slave tarato
RT_TARAS: R_TRIG;
#defcom RT_SLVQT.Q Imp. fine ciclo taratura gantry
RT_SLVQT: R_TRIG;
#defcom T_WSTREF.Q Fine attesa stop asse dopo taratura
T_WSTREF: TON;
#defcom T_ALL.Q Allineamento slave completato
T_ALL: TON ;

GANTFB: CN_GANTRY;
TAR_X1: CYC_HOMING;
TAR_X2: CYC_HOMING;
POS_X1: AX_POSIZ;
POS_X2: AX_POSIZ;
PRS_X2: AX_PRESET;
END_VAR

PATH %ax[xNSlave]                  ** Numero asse slave

LD   BAO_GTRYLINK                  ** ra3.17  Accoppiamento Gantry attivo
ST   GantryOnS                     ** Gantry attivo su asse slave

LD   BAO_ALLM                      ** ra3.15  Asse in Allarme
ST   AlarmS                        ** Allarme su asse slave

LD   BAO_AFET                      ** ra3.0  Asse fermo teorico
ST   AxFermoS                      ** Asse slave fermo

LD   BAO_TARA                      ** ra3.14  Asse tarato
ST   AxTaratoS                     ** Asse slave tarato

LD   BAO_ISO_NULLO                 ** ra19.0 Stato NULLO all'interno del canale
ST   IsoNullS                      ** Asse slave in ISO nullo

LD   AO_QUOTA                      ** ra4  Quota asse
ST   PosSlave                      ** Quota attuale asse slave

LD   %ra10
EQ   0
ST   CodeLibereSlave               ** Nessun comando su coda slave

PATH %ax[xNMaster]                 ** Numero asse master
PATH %gantry[AP_AXNGANTRY]         ** pa47 Indice tabella gantry

CAL  RT_TARAM(CLK=BAO_TARA)        ** ra3.14  Asse tarato

* Consensi gantry attivo/inattivo

LDN  BAO_GTRYLINK                  ** ra3.17  Accoppiamento Gantry attivo
ANDN GantryOnS                     ** Gantry attivo su asse slave
ST   yGantryOff                    ** Accoppiamento gantry non attivo

LD   BAO_GTRYLINK                  ** ra3.17  Accoppiamento Gantry attivo
AND  GantryOnS                     ** Gantry attivo su asse slave
ST   yGantryOn                     ** Accoppiamento gantry attivo

* Tipo di taratura del gantry

LD   GDAT6                         ** Gdat6 Tipo taratura (0=standard, 1=con 1 finecorsa)
EQ   1
ST   Ref1LS                        ** Ciclo taratura con 1 finecorsa

LD   RT_TARAM.Q                    ** Imp. asse master tarato
S    MemZeroM                      ** Mem. asse master tarato

LDN  yRefM                         ** Richiesta ciclo zero su asse master
R    MemZeroM                      ** Mem. asse master tarato

LD   %ra10
EQ   0
AND  MemZeroM                      ** Mem. asse master tarato
AND  xExtCmd                       ** Selezione comandi REF-JOG esterni (da canale)
OR   TAR_X1.yax_ENDOK
ST   EndZeroM                      ** Ciclo taratura asse master effettuato

CAL  RT_TARAS(CLK=AxTaratoS)       ** Asse slave tarato

LD   RT_TARAS.Q                    ** Imp. asse slave tarato
S    MemZeroS                      ** Mem. asse slave tarato

LDN  yRefS                         ** Richiesta ciclo zero su asse slave
R    MemZeroS                      ** Mem. asse slave tarato

LD   MemZeroS                      ** Mem. asse slave tarato
AND  xExtCmd                       ** Selezione comandi REF-JOG esterni (da canale)
AND  CodeLibereSlave               ** Nessun comando su coda slave
OR   TAR_X2.yax_ENDOK
ST   EndZeroS                      ** Ciclo taratura asse slave effettuato

* Ciclo taratura con assi gantry

LD   xRefCycle                     ** Comando esecuzione ciclo di taratura
ANDN yOnOff                        ** Comando aggancio-sgancio in corso
ANDN CPASga                        ** Ciclo allinea gantry: sgancio gantry
ANDN CARSga                        ** Ciclo allinea al ripristino emergenza: sgancio gantry
S    CTGPreset                     ** Ciclo tara gantry: preset iniziale

LD   PRS_X2.yax_ENDOK
OR   yGantryOn                     ** Accoppiamento gantry attivo
AND  CTGPreset                     ** Ciclo tara gantry: preset iniziale
S    CTGFirstAgg                   ** Ciclo tara gantry: primo aggancio gantry

LD   yGantryOn                     ** Accoppiamento gantry attivo
AND  GANTFB.ycn_ENDOK
AND  CTGFirstAgg                   ** Ciclo tara gantry: primo aggancio gantry
S    CTGZeroM                      ** Ciclo tara gantry: ricerca zero su asse master

LD   EndZeroM                      ** Ciclo taratura asse master effettuato
AND  CTGZeroM                      ** Ciclo tara gantry: ricerca zero su asse master
ANDN Ref1LS                        ** Ciclo taratura con 1 finecorsa
S    CTGSlaveAgg                   ** Ciclo tara gantry: aggancio gantry slave-master

LD   yGantryOn                     ** Accoppiamento gantry attivo
AND  GANTFB.ycn_ENDOK
AND  CTGSlaveAgg                   ** Ciclo tara gantry: aggancio gantry slave-master
S    CTGZeroS                      ** Ciclo tara gantry: ricerca zero su asse slave

LD   EndZeroS                      ** Ciclo taratura asse slave effettuato
AND  CTGZeroS                      ** Ciclo tara gantry: ricerca zero su asse slave
OR   (
LD   EndZeroM                      ** Ciclo taratura asse master effettuato
AND  CTGZeroM                      ** Ciclo tara gantry: ricerca zero su asse master
AND  Ref1LS                        ** Ciclo taratura con 1 finecorsa
)
S    CTGLastSga                    ** Ciclo tara gantry: ultimo sgancio gantry

LD   yGantryOff                    ** Accoppiamento gantry non attivo
AND  CTGLastSga                    ** Ciclo tara gantry: ultimo sgancio gantry
ANDN xZeroSetup                    ** Esclude allineamento a fine taratura
S    CTGAllin                      ** Ciclo tara gantry: posiziona slave alla quota master

LD   T_ALL.Q                       ** Allineamento slave completato
AND  CTGAllin                      ** Ciclo tara gantry: posiziona slave alla quota master
S    CTGLastAgg                    ** Ciclo tara gantry: ultimo aggancio gantry

LD   yGantryOn                     ** Accoppiamento gantry attivo
AND  CTGLastAgg                    ** Ciclo tara gantry: ultimo aggancio gantry
AND  xParkCycle                    ** Abilita ciclo parcheggio a fine taratura
S    CTGPark                       ** Ciclo tara gantry: parcheggio gantry

LDN  xRefCycle                     ** Comando esecuzione ciclo di taratura
R    CTGPreset                     ** Ciclo tara gantry: preset iniziale
R    CTGFirstAgg                   ** Ciclo tara gantry: primo aggancio gantry
R    CTGZeroM                      ** Ciclo tara gantry: ricerca zero su asse master
R    CTGSlaveAgg                   ** Ciclo tara gantry: aggancio gantry slave-master
R    CTGZeroS                      ** Ciclo tara gantry: ricerca zero su asse slave
R    CTGLastSga                    ** Ciclo tara gantry: ultimo sgancio gantry
R    CTGAllin                      ** Ciclo tara gantry: posiziona slave alla quota master
R    CTGLastAgg                    ** Ciclo tara gantry: ultimo aggancio gantry
R    CTGPark                       ** Ciclo tara gantry: parcheggio gantry

LD   yGantryOn                     ** Accoppiamento gantry attivo
AND  CTGLastAgg                    ** Ciclo tara gantry: ultimo aggancio gantry
ANDN xParkCycle                    ** Abilita ciclo parcheggio a fine taratura
OR   (
LD   POS_X1.yax_ENDOK
AND  CTGPark                       ** Ciclo tara gantry: parcheggio gantry
)
OR   (
LD   yGantryOff                    ** Accoppiamento gantry non attivo
AND  CTGLastSga                    ** Ciclo tara gantry: ultimo sgancio gantry
AND  xZeroSetup                    ** Esclude allineamento a fine taratura
)
ST   yEndCycRef                    ** Fine ciclo taratura gantry

CAL  T_WSTREF(IN=CTGAllin, PT=1000) ** Ciclo tara gantry: posiziona slave alla quota master

LD   AO_QUOTA                      ** ra4  Quota asse
SUB  PosSlave                      ** Quota attuale asse slave
ABS
GE   GDAT3                         ** Gdat3 Tolleranza Allarme REF
AND  T_WSTREF.Q                    ** Fine attesa stop asse dopo taratura
S    yRefAlarm                     ** Allarme allineamento durante ciclo zero

LD   xReset                        ** Reset comandi gantry
R    yRefAlarm                     ** Allarme allineamento durante ciclo zero

* Ciclo preset o allineamento slave alla quota del master

LD   xReqPreset                    ** Richiesta preset slave alla quota del master
OR   xReqAllin                     ** Richiesta allineamento slave alla quota del master
ANDN yOnOff                        ** Comando aggancio-sgancio in corso
ANDN CTGPreset                     ** Ciclo tara gantry: preset iniziale
S    CPASga                        ** Ciclo allinea gantry: sgancio gantry

LD   yGantryOff                    ** Accoppiamento gantry non attivo
AND  CPASga                        ** Ciclo allinea gantry: sgancio gantry
S    CPAExec                       ** Ciclo allinea gantry: esegue preset o allineamento

LD   PRS_X2.yax_ENDOK
AND  xReqPreset                    ** Richiesta preset slave alla quota del master
OR   (
LD   T_ALL.Q                       ** Allineamento slave completato
AND  xReqAllin                     ** Richiesta allineamento slave alla quota del master
)
AND  CPAExec                       ** Ciclo allinea gantry: esegue preset o allineamento
S    CPARiagg                      ** Ciclo allinea gantry: riaggancio gantry

LDN  xReqPreset                    ** Richiesta preset slave alla quota del master
ANDN xReqAllin                     ** Richiesta allineamento slave alla quota del master
R    CPASga                        ** Ciclo allinea gantry: sgancio gantry
R    CPAExec                       ** Ciclo allinea gantry: esegue preset o allineamento
R    CPARiagg                      ** Ciclo allinea gantry: riaggancio gantry

LD   yGantryOn                     ** Accoppiamento gantry attivo
AND  CPARiagg                      ** Ciclo allinea gantry: riaggancio gantry
ST   yEndPrAll                     ** Fine preset o allineamento slave a quota master

* Memoria eseguito ciclo setup: il ciclo setup attiva il bit di asse tarato,
* ma le quote di taratura degli assi non sono ancora state messe a punto,
* quindi debbo bloccare l'allineamento automatico dopo emergenza finch�
* non avr� eseguito un ciclo di taratura valido.

LD   xZeroSetup                    ** Esclude allineamento a fine taratura
AND  yEndCycRef                    ** Fine ciclo taratura gantry
S    MemSetupDone                  ** Mem. eseguito ciclo setup

LDN  xZeroSetup                    ** Esclude allineamento a fine taratura
AND  yEndCycRef                    ** Fine ciclo taratura gantry
R    MemSetupDone                  ** Mem. eseguito ciclo setup

* Abilita allineamento gantry dopo emergenza: se attivo, allinea,
* se inattivo, effettua il preset dello slave.
* Serve per evitare il riallineamento automatico al ripristino da emergenza
* finch� non � stato eseguito un ciclo di taratura valido,
* altrimenti si rischia di allineare su quote errate e danneggiare il gantry.

LDN  MemSetupDone                  ** Mem. eseguito ciclo setup
AND  AxTaratoS                     ** Asse slave tarato
AND  BAO_TARA                      ** ra3.14  Asse tarato
ST   AllDopoEmer                   ** Abilita allineamento gantry dopo emergenza

* Ciclo allineamento slave al ripristino da emergenza

LD   xEmer                         ** Condizioni di emergenza che forzano l'apertura del gantry
AND  BAO_AFET                      ** ra3.0  Asse fermo teorico
AND  AxFermoS                      ** Asse slave fermo
OR   ON_ONE_SCAN                   ** PLCFLAGS.8  Flag on alla prima scansione PLC
S    CARSga                        ** Ciclo allinea al ripristino emergenza: sgancio gantry

LDN  xEmer                         ** Condizioni di emergenza che forzano l'apertura del gantry
ANDN xReset                        ** Reset comandi gantry
AND  yGantryOff                    ** Accoppiamento gantry non attivo
AND  CARSga                        ** Ciclo allinea al ripristino emergenza: sgancio gantry
AND (
LD   PosMaster                     ** Quota attuale asse master
SUB  PosSlave                      ** Quota attuale asse slave
ABS
LT   GDAT2                         ** Gdat2 Tolleranza Allarme
)
S    CARAllin                      ** Ciclo allinea al ripristino emergenza: esegue allineamento

LD   T_ALL.Q                       ** Allineamento slave completato
OR   PRS_X2.yax_ENDOK
AND  CARAllin                      ** Ciclo allinea al ripristino emergenza: esegue allineamento
S    CARRiagg                      ** Ciclo allinea al ripristino emergenza: riaggancio gantry

LD   yGantryOn                     ** Accoppiamento gantry attivo
AND  CARRiagg                      ** Ciclo allinea al ripristino emergenza: riaggancio gantry
OR   (
LD   xEmer                         ** Condizioni di emergenza che forzano l'apertura del gantry
AND  CARAllin                      ** Ciclo allinea al ripristino emergenza: esegue allineamento
)
R    CARSga                        ** Ciclo allinea al ripristino emergenza: sgancio gantry
R    CARAllin                      ** Ciclo allinea al ripristino emergenza: esegue allineamento
R    CARRiagg                      ** Ciclo allinea al ripristino emergenza: riaggancio gantry

LD   CARSga                        ** Ciclo allinea al ripristino emergenza: sgancio gantry
ST   yAlPr                         ** Comando allineamento-preset dopo ripristino emergenza in corso

* FB attiva/disattiva GANTRY

LD   BCO_CANREADY                  ** rc8.2  Canale Ready
ANDN xReset                        ** Reset comandi gantry
ST   BCI_PLCREQ                    ** cnfb23.28 Richiesta gestione processo da PLC
ST   GANTFB.xcn_ENABLE       * abilita FB

LD   CTGFirstAgg                   ** Ciclo tara gantry: primo aggancio gantry
ANDN CTGZeroM                      ** Ciclo tara gantry: ricerca zero su asse master
OR   (
LD   CTGSlaveAgg                   ** Ciclo tara gantry: aggancio gantry slave-master
ANDN CTGZeroS                      ** Ciclo tara gantry: ricerca zero su asse slave
)
ST   ForzAggancio                  ** Cond. forzamento aggancio gantry (anche se lo � gi�)

LD   ForzAggancio                  ** Cond. forzamento aggancio gantry (anche se lo � gi�)
OR   CTGLastAgg                    ** Ciclo tara gantry: ultimo aggancio gantry
OR   CPARiagg                      ** Ciclo allinea gantry: riaggancio gantry
OR   CARRiagg                      ** Ciclo allinea al ripristino emergenza: riaggancio gantry
OR   xReqAggancio                  ** Richiesta aggancio gantry
S    MemAggancio                   ** Mem. aggancio gantry

LD   CTGLastSga                    ** Ciclo tara gantry: ultimo sgancio gantry
ANDN CTGLastAgg                    ** Ciclo tara gantry: ultimo aggancio gantry
OR   (
LD   CPASga                        ** Ciclo allinea gantry: sgancio gantry
ANDN CPAExec                       ** Ciclo allinea gantry: esegue preset o allineamento
)
OR   (
LD   CARSga                        ** Ciclo allinea al ripristino emergenza: sgancio gantry
ANDN CARAllin                      ** Ciclo allinea al ripristino emergenza: esegue allineamento
)
OR   xReqSgancio                   ** Richiesta sgancio gantry
OR   BAO_GTRYALRM                  ** ra6.19 Allarme per disallineamento gantry
R    MemAggancio                   ** Mem. aggancio gantry

LD   MemAggancio                   ** Mem. aggancio gantry
ANDN yGantryOn                     ** Accoppiamento gantry attivo
OR   ForzAggancio                  ** Cond. forzamento aggancio gantry (anche se lo � gi�)
* Controllo lo stato ISO nullo perch� se tento di agganciare il gantry al volo
* mi d� errore, in particolare durante la taratura in cui in certi casi
* lo slave toglieva il bit di gantry agganciato.
AND  BAO_ISO_NULLO                 ** ra19.0 Stato NULLO all'interno del canale
AND  IsoNullS                      ** Asse slave in ISO nullo
ANDN xEmer                         ** Condizioni di emergenza che forzano l'apertura del gantry
OR   (
LDN  MemAggancio                   ** Mem. aggancio gantry
ANDN yGantryOff                    ** Accoppiamento gantry non attivo
)
* Se l'aggancio va in allarme disallineamento, attende un attimo
* prima di sganciare per sincronizzare il blocco di aggancio-sgancio
AND  (
LDN  BAO_GTRYALRM                  ** ra6.19 Allarme per disallineamento gantry
ANDN GANTFB.ycn_ENDOK
)
AND  GANTFB.xcn_ENABLE       * abilita FB
ST   yOnOff                        ** Comando aggancio-sgancio in corso

LD   yOnOff                        ** Comando aggancio-sgancio in corso
AND  GANTFB.ycn_READY
ANDN GANTFB.ycn_ENDOK
ANDN GANTFB.ycn_ENDERR
ANDN xAuxBusy                      ** Canale ausiliario impegnato
ST   GANTFB.xcn_START

LDN  yOnOff                        ** Comando aggancio-sgancio in corso
ST   GANTFB.xcn_CLEAR

LD   MemAggancio                   ** Mem. aggancio gantry
ST   GANTFB.xcn_ONOFF

LD   ALWAYS_ONE                    ** PLCFLAGS.1  Flag sempre stato on
ST   GANTFB.xcn_COPY

LD   AP_AXNGANTRY                  ** pa47 Indice tabella gantry
ST   GANTFB.xcn_INDEX

LD   xNMaster                      ** Numero asse master
ST   GANTFB.xcn_MASTER

LD   CTGSlaveAgg                   ** Ciclo tara gantry: aggancio gantry slave-master
ANDN CTGAllin                      ** Ciclo tara gantry: posiziona slave alla quota master
JMPCN GNT_SLAVE

LD   xNSlave                       ** Numero asse slave
ST   GANTFB.xcn_MASTER

GNT_SLAVE:

LD   CTGFirstAgg                   ** Ciclo tara gantry: primo aggancio gantry
ANDN CTGLastSga                    ** Ciclo tara gantry: ultimo sgancio gantry
OR   xNoAlarm                      ** Esclude allarme massimo disallineamento
ST   GANTFB.xcn_REFTOLL

CAL  GANTFB

LD   GANTFB.ycn_ERRCODE
ST   ycn_ERRCODE                   ** Function-Block error code

* Comando output per richiesta comandi esterni

LD   CTGZeroM                      ** Ciclo tara gantry: ricerca zero su asse master
ANDN CTGSlaveAgg                   ** Ciclo tara gantry: aggancio gantry slave-master
ANDN CTGLastSga                    ** Ciclo tara gantry: ultimo sgancio gantry
AND  xExtCmd                       ** Selezione comandi REF-JOG esterni (da canale)
ST   yRefM                         ** Richiesta ciclo zero su asse master

LD   CTGZeroS                      ** Ciclo tara gantry: ricerca zero su asse slave
ANDN CTGLastSga                    ** Ciclo tara gantry: ultimo sgancio gantry
AND  xExtCmd                       ** Selezione comandi REF-JOG esterni (da canale)
ST   yRefS                         ** Richiesta ciclo zero su asse slave

LD   CTGPreset                     ** Ciclo tara gantry: preset iniziale
ANDN xExtCmd                       ** Selezione comandi REF-JOG esterni (da canale)
OR   CTGAllin                      ** Ciclo tara gantry: posiziona slave alla quota master
ANDN CTGLastAgg                    ** Ciclo tara gantry: ultimo aggancio gantry
OR   (
LD   CTGPreset                     ** Ciclo tara gantry: preset iniziale
ANDN CTGFirstAgg                   ** Ciclo tara gantry: primo aggancio gantry
)
OR   (
LD   CPAExec                       ** Ciclo allinea gantry: esegue preset o allineamento
ANDN CPARiagg                      ** Ciclo allinea gantry: riaggancio gantry
)
OR   (
LD   CARAllin                      ** Ciclo allinea al ripristino emergenza: esegue allineamento
ANDN CARRiagg                      ** Ciclo allinea al ripristino emergenza: riaggancio gantry
)
OR   CTGPark                       ** Ciclo tara gantry: parcheggio gantry
ANDN yRefM                         ** Richiesta ciclo zero su asse master
ANDN yRefS                         ** Richiesta ciclo zero su asse slave
ST   yGrant                        ** Richiesta comando assi da PLC

* Comandi asse master

* Taratura asse con ricerca tacca

LD   CTGZeroM                      ** Ciclo tara gantry: ricerca zero su asse master
ANDN CTGSlaveAgg                   ** Ciclo tara gantry: aggancio gantry slave-master
ANDN CTGLastSga                    ** Ciclo tara gantry: ultimo sgancio gantry
ANDN xExtCmd                       ** Selezione comandi REF-JOG esterni (da canale)
ANDN xReset                        ** Reset comandi gantry
ST   TAR_X1.xax_ENABLE

LDN  TAR_X1.xax_ENABLE
ST   TAR_X1.xax_CLEAR

LD   TAR_X1.xax_ENABLE
AND  TAR_X1.yax_READY
ANDN TAR_X1.yax_ENDOK
ANDN TAR_X1.yax_ENDERR
ST   TAR_X1.xax_START

CAL  TAR_X1

* Posizionamento asse

LD   CTGPark                       ** Ciclo tara gantry: parcheggio gantry
ANDN xReset                        ** Reset comandi gantry
ST   POS_X1.xax_ENABLE

LDN  POS_X1.xax_ENABLE
ST   POS_X1.xax_CLEAR

LD   POS_X1.xax_ENABLE
AND  POS_X1.yax_READY
ANDN POS_X1.yax_ENDOK
ANDN POS_X1.yax_ENDERR
ST   POS_X1.xax_START

LD   AP_PARKQTA                    ** pa31 Quota di parcheggio
ST   POS_X1.xax_QUOTA

LD   xParkSpeed                    ** Velocit� di parcheggio
EQ   0
JMPC PARK_VELMAN

LD   xParkSpeed                    ** Velocit� di parcheggio
ST   POS_X1.xax_VEL

JMP  PARK_VELEND

PARK_VELMAN:

LD   %pa60
ST   POS_X1.xax_VEL

PARK_VELEND:

CAL  POS_X1

LD   AO_QUOTA                      ** ra4  Quota asse
ST   PosMaster                     ** Quota attuale asse master

* Comandi asse slave

PATH %ax[xNSlave]                  ** Numero asse slave

* Taratura asse con ricerca tacca

LD   CTGZeroS                      ** Ciclo tara gantry: ricerca zero su asse slave
ANDN CTGLastSga                    ** Ciclo tara gantry: ultimo sgancio gantry
ANDN xExtCmd                       ** Selezione comandi REF-JOG esterni (da canale)
ANDN xReset                        ** Reset comandi gantry
ST   TAR_X2.xax_ENABLE

LDN  TAR_X2.xax_ENABLE
ST   TAR_X2.xax_CLEAR

LD   TAR_X2.xax_ENABLE
AND  TAR_X2.yax_READY
ANDN TAR_X2.yax_ENDOK
ANDN TAR_X2.yax_ENDERR
ST   TAR_X2.xax_START

CAL  TAR_X2

* Posizionamento asse

LD   T_WSTREF.Q                    ** Fine attesa stop asse dopo taratura
ANDN CTGLastAgg                    ** Ciclo tara gantry: ultimo aggancio gantry
ANDN yRefAlarm                     ** Allarme allineamento durante ciclo zero
OR   (
LD   CPAExec                       ** Ciclo allinea gantry: esegue preset o allineamento
ANDN CPARiagg                      ** Ciclo allinea gantry: riaggancio gantry
AND  xReqAllin                     ** Richiesta allineamento slave alla quota del master
)
OR   (
LD   CARAllin                      ** Ciclo allinea al ripristino emergenza: esegue allineamento
ANDN CARRiagg                      ** Ciclo allinea al ripristino emergenza: riaggancio gantry
AND  AllDopoEmer                   ** Abilita allineamento gantry dopo emergenza
)
ANDN xReset                        ** Reset comandi gantry
ST   POS_X2.xax_ENABLE

LDN  POS_X2.xax_ENABLE
ST   POS_X2.xax_CLEAR

LD   POS_X2.xax_ENABLE
AND  POS_X2.yax_READY
ANDN POS_X2.yax_ENDOK
ANDN POS_X2.yax_ENDERR
ST   POS_X2.xax_START

LD   PosMaster                     ** Quota attuale asse master
ST   POS_X2.xax_QUOTA

LD   AP_VELMICRO                   ** pa19 Velocit� ricerca micro in taratura
ST   POS_X2.xax_VEL

CAL  POS_X2

CAL  T_ALL(IN=POS_X2.yax_ENDOK, PT=AP_TIMERTOLL) ** pa8 Preset timer tolleranza

* Preset asse

LD   CPAExec                       ** Ciclo allinea gantry: esegue preset o allineamento
ANDN CPARiagg                      ** Ciclo allinea gantry: riaggancio gantry
AND  xReqPreset                    ** Richiesta preset slave alla quota del master
OR   (
LD   CTGPreset                     ** Ciclo tara gantry: preset iniziale
ANDN CTGFirstAgg                   ** Ciclo tara gantry: primo aggancio gantry
)
OR   (
LD   CARAllin                      ** Ciclo allinea al ripristino emergenza: esegue allineamento
ANDN CARRiagg                      ** Ciclo allinea al ripristino emergenza: riaggancio gantry
ANDN AllDopoEmer                   ** Abilita allineamento gantry dopo emergenza
)
ANDN xReset                        ** Reset comandi gantry
ST   PRS_X2.xax_ENABLE

LDN  PRS_X2.xax_ENABLE
ST   PRS_X2.xax_CLEAR

LD   PRS_X2.xax_ENABLE
AND  PRS_X2.yax_READY
ANDN PRS_X2.yax_ENDOK
ANDN PRS_X2.yax_ENDERR
ST   PRS_X2.xax_START

LD   PosMaster                     ** Quota attuale asse master
ST   PRS_X2.xax_QUOTA

CAL  PRS_X2

LD   PRS_X2.xax_ENABLE
ST   yPresetReq                    ** Richesta preset asse Slave

* Procedura modifica quota taratura slave alla fine del ciclo di zero setup.
* Somma alla quota di zero slave la differenza tra i due assi.

LD   yEndCycRef                    ** Fine ciclo taratura gantry
ST   RT_SLVQT.CLK

CAL  RT_SLVQT

LD   RT_SLVQT.Q                    ** Imp. fine ciclo taratura gantry
AND  xZeroSetup                    ** Esclude allineamento a fine taratura
AND  xAutZeroSetup                 ** Modifica automatica quota taratura a fine setup
JMPCN END_SLVQT

LD   PosMaster                     ** Quota attuale asse master
SUB  AO_QUOTA                      ** ra4  Quota asse
ADD  QTA_TARA_SLAVE                ** pa18 Quota di taratura asse
ST   QTA_TARA_SLAVE                ** pa18 Quota di taratura asse

END_SLVQT:

END_FUNCTION_BLOCK

* FB Comando segnali modulo VRTC
VAR_IN_OUT
VRTC_CR0           AT %VrdwCtrlRegister0;   * VRTC control register 0
VRTC_CR1           AT %VrdwCtrlRegister1;   * VRTC control register 1
VRTC_AR0           AT %VrdwAckRegister0;    * VRTC acknowledge register 0
VRTC_AR1           AT %VrdwAckRegister1;    * VRTC acknowledge register 1
VRTC_SR0           AT %VrdwStatRegister0;   * VRTC status register 0
VRTC_SR1           AT %VrdwStatRegister1;   * VRTC status register 1
VRTC_SIMOFF_SET    AT %VrSim_Q_OffsetSet;   * VRTC simulation offset set
VRTC_SIMOFF_CUR    AT %VrEq_Q_OffsetCur;    * VRTC simulation offset current
VRTC_SETPOINT      AT %VrU_Setpoint;        * VRTC setpoint
VRTC_SENSOR_IN     AT %VrSensorInput;       * VRTC Sensor Input

VRTC_POS_UPLIM     AT %VrLimM_Q_U;          * VRTC mandatory position upper limit (mm)
VRTC_POS_LWLIM     AT %VrLimM_Q_L;          * VRTC mandatory position lower limit (mm)
VRTC_VEL_UPLIM     AT %VrLimM_Q_D_U;        * VRTC mandatory velocity upper limit
VRTC_VEL_LWLIM     AT %VrLimM_Q_D_D;        * VRTC mandatory velocity lower limit
VRTC_ACC_UPLIM     AT %VrLimM_Q_DD_U;       * VRTC mandatory acceleration upper limit (mm)
VRTC_ACC_LWLIM     AT %VrLimM_Q_DD_D;       * VRTC mandatory acceleration lower limit (mm)
VRTC_KPGAIN        AT %VrKpGain;            * VRTC Kp gain [[mm/s]/U]
VRTC_NON_LINEAR_MODE AT %VrNonLinearMode;     * VRTC non-linear regulation mode
VRTC_KP_TABLE      AT %VrKpTransPtr;        * VRTC Kp trans-characteristics table index
VRTC_KP_TABLE_MUL  AT %VrKpTransMul;        * VRTC Kp trans-characteristics table multiplier
VRTC_SLIDING_DECEL AT %VrSlidingDecel;      * VRTC sliding mode deceleration [mm/s�]
VRTC_DB_POS        AT %VrU_DbPos;           * VRTC positive deadband
VRTC_DB_NEG        AT %VrU_DbNeg;           * VRTC negative deadband
VRTC_CUTOFF        AT %VrFilter_FreqHz;     * VRTC Filter cutoff frequency [Hz]
VRTC_DAMPING       AT %VrFilter_DampingC;   * VRTC Damping filter
VRTC_SIM_FADER     AT %VrSimFadingTime;     * VRTC Simulation Xfade time [ms]
VRTC_TRIG_VEL_UP   AT %VrLimL_Flt_Q_D_U;    * VRTC Lock trigger velocity Up
VRTC_TRIG_VEL_LW   AT %VrLimL_Flt_Q_D_D;    * VRTC Lock trigger velocity Down
VRTC_TRIG_ACC      AT %VrLimL_Flt_Q_DD;     * VRTC Lock trigger acceleration
END_VAR

* VRTC_EX FB SECTION
*=========================================================================

VAR_IN_OUT
VRTC_VECTOR_SELECT  AT %VrVectorSelect;      * VRTC vector select
VRTC_SIM_OFFSET_SET AT %VrSim_Q_OffsetSet;   * VRTC simulation offset set
VRTC_SIM_OFFSET_CUR AT %VrEq_Q_OffsetCur;    * VRTC simulation offset cur
VRTC_FLT_Q          AT %VrMon_Q_Flt_Q;       * VRTC contribution
END_VAR

FUNCTION_BLOCK VRTC_EX

VAR_INPUT
xVectorSelect: DWORD; * Vector select
xReset: BOOL; * Reset
xSimul: BOOL; * Simulazione
xMoveToTarget: BOOL; * Richiesta movimento su target
xResPosInt: BOOL; * Reset position integrator
xPosLimDisab: BOOL; * Disable mandatory position limit
xDeOverlapEnab: BOOL; * Enable de-overlap
xErrorAmpEnab: BOOL; * Enable error amplifier
xMLonlyClampFilterIn:   BOOL;
xMLonlyClampFilterInDot: BOOL;

xSimOffsetSet: DWORD; * VRTC simulation offset set
xSetPoint: DWORD; * VRTC set point
xSensorIn: DWORD; * Sensor Input

xUpPosLimit: DWORD; * Mandatory upper position limit
xLwPosLimit: DWORD; * Mandatory lower position limit
xVelLimitUp: DWORD; * Upward Mandatory velocity limit
xVelLimitDown: DWORD; * Downward Mandatory velocity limit
xAccLimitUp: DWORD; * Upward Mandatory velocity limit
xAccLimitDown: DWORD; * Downward Mandatory velocity limit
xKpGain: DWORD; * Kp gain [[mm/s]/U]
xKpTransPtr:  DWORD; * Kp trans-characteristics table index
xKpTransMul:  DWORD; * Kp trans-characteristics table multiplier (<>0 == enable)
xSlidingDecel:  DWORD; * Sliding mode deceleration [mm/s�] (<>0 == enable)
xDbPos:  DWORD; * positive deadband
xDbNeg:  DWORD; * negative deadband
xFilterCutOff: DWORD; * Filter cutoff frequency [Hz]
xFilterDamping: DWORD; * Filter Damping Coefficient
xSimFadingTime:  DWORD; * Simulation Xfade time [ms]
xLockVelLimitUp:  DWORD; * Lock trigger velocity Up
xLockVelLimitDown:  DWORD; * Lock trigger velocity Down
xLockAccLimit:  DWORD; * Lock trigger acceleration

END_VAR

VAR_OUTPUT
yBusy: BOOL; * Comando VRTC in corso
ySignalLock: BOOL; * VRTC locked
ySimOffsetCur: DWORD; * last VRTC simulation offset
yFltQ: DWORD; * VRTC contribution
END_VAR

VAR
#defcom TR_VRTSIM.Q Simulazione
TR_VRTSIM: TRIG;
#defcom TR_VRTRST.Q Reset VRTC
TR_VRTRST: TRIG;
#defcom TR_VRTRPI.Q Imp. reset position integrator
TR_VRTRPI: TRIG;
#defcom TR_VRTPLD.Q Imp. disable mandatory position limit
TR_VRTPLD: TRIG;
#defcom TR_DEOVER.Q Enable de-overlap
TR_DEOVER: TRIG;
#defcom TR_ERRAMP.Q Enable error amplifier
TR_ERRAMP: TRIG;
TR_MLonlyClamp: TRIG;
TR_MLonlyClampDot: TRIG;

CtrReg0: DWORD; * Appoggio control register 0
CtrReg1: DWORD; * Appoggio control register 1
DwCrtReg1: DWORD; * Appoggio DW control register 1
AckReg0: DWORD; * Appoggio ACK register 0
AckReg1: DWORD; * Appoggio ACK register 1
StatReg0: DWORD; * Appoggio status register 0
StatReg1: DWORD; * Appoggio status register 1

PrevSimOffsetSet: DWORD; * Valore precedente simulation offset set

PrevUpPosLim:       DWORD; * Previous mandatory upper position limit
PrevLwPosLim:       DWORD; * Previous mandatory lower position limit
PrevUpVelLim:       DWORD; * Previous Up mandatory velocity limit
PrevDnVelLim:       DWORD; * Previous Down mandatory velocity limit
PrevUpAccLim:       DWORD; * Previous Up mandatory acceleration limi
PrevDnAccLim:       DWORD; * Previous Down mandatory acceleration limit
PrevKpGain:         DWORD; * Previous Kp gain
PrevKpTransPtr:     DWORD; * Previous Kp trans-characteristics table index
PrevKpTransMul:     DWORD; * Previous Kp trans-characteristics table multiplier (<>0 == enable)
PrevSlidingDecel:   DWORD; * Previous sliding mode deceleration [mm/s�] (<>0 == enable)
PrevDbPos:          DWORD; * Previous positive deadband
PrevDbNeg:          DWORD; * Previous negative deadband
PrevFilterCutOff:   DWORD; * Previous Filter cutoff frequency
PrevFilterDamping:  DWORD; * Previous filter damping value
PrevSimFadingTime:  DWORD; * Previous Simulation Xfade time [ms]
PrevLockVelLimitUp: DWORD; * Previous Lock trigger velocity Up
PrevLockVelLimitDn: DWORD; * Previous Lock trigger velocity Down
PrevLockAccLimit:   DWORD; * Previous Lock trigger acceleration
PrevSetpoint:       DWORD; * Previous Setpoint
END_VAR

* Acknowledge register 0

LD      VRTC_AR0                   ** VRTC acknowledge register 0
ST      AckReg0                    ** Appoggio ACK register 0

* Acknowledge register 1

LD      VRTC_AR1                   ** VRTC acknowledge register 1
ST      AckReg1                    ** Appoggio ACK register 1

* Vector Select

LD      xVectorSelect
ST      VRTC_VECTOR_SELECT

* Control register 0

LD      %PLCFLAGS.1
ST      CtrReg0.9           * Enable velocity feed-forward
ST      CtrReg0.24          * Auxiliary signal #0 (registers update)

* Master reset

LD      xReset                     ** Reset
ST      CtrReg0.0           * Master reset

* Master enable

LDN     xReset                     ** Reset
ST      CtrReg0.1           * Master enable

* Enable error amplifier

LD      xErrorAmpEnab              ** Enable error amplifier
ST      CtrReg0.2           * Enable error amplifier

* Enable off-sensor simulation

LD      xSimul                     ** Simulazione
ST      CtrReg0.3           * Enable off-sensor simulation

* Reset position integrator

LD      xResPosInt                 ** Reset position integrator
ST      CtrReg0.5           * Reset position integrator

* Enable de-overlap

LD      xDeOverlapEnab             ** Enable de-overlap
ST      CtrReg0.18          * Enable de-overlap

* Enable mandatory position limit

LDN     xPosLimDisab               ** Disable mandatory position limit
ANDN    xResPosInt                 ** Reset position integrator
ANDN    xReset                     ** Reset
ST      CtrReg1.12          * Enable mandatory position limit

* Mandatory position limit

LD      xUpPosLimit                ** Mandatory upper position limit
ST      VRTC_POS_UPLIM             ** VRTC mandatory position upper limit (mm)
LD      xLwPosLimit                ** Mandatory lower position limit
ST      VRTC_POS_LWLIM             ** VRTC mandatory position lower limit (mm)

* Mandatory velocity limit

LD      xVelLimitUp                ** Upward Mandatory velocity limit
ST      VRTC_VEL_UPLIM             ** VRTC mandatory velocity upper limit
LD      xVelLimitDown              ** Downward Mandatory velocity limit
ST      VRTC_VEL_LWLIM             ** VRTC mandatory velocity lower limit

LD      xVelLimitUp                ** Upward Mandatory velocity limit
NE      0
OR (
LD      xVelLimitDown              ** Downward Mandatory velocity limit
NE      0
)
ST      CtrReg1.13                    * Enable mandatory velocity limit

* Mandatory acceleration limit

LD      xAccLimitUp                ** Upward Mandatory velocity limit
ST      VRTC_ACC_UPLIM             ** VRTC mandatory acceleration upper limit (mm)
LD      xAccLimitDown              ** Downward Mandatory velocity limit
ST      VRTC_ACC_LWLIM             ** VRTC mandatory acceleration lower limit (mm)

LD      xAccLimitUp                ** Upward Mandatory velocity limit
NE      0
OR (
LD      xAccLimitDown              ** Downward Mandatory velocity limit
NE      0
)
ST      CtrReg1.14                    * Enable mandatory acceleration limit

* Kp gain

LD      xKpGain                    ** Kp gain [[mm/s]/U]
ST      VRTC_KPGAIN                ** VRTC Kp gain [[mm/s]/U]

* Kp trans-characteristics table

LD      xKpTransPtr                ** Kp trans-characteristics table index
ST      VRTC_KP_TABLE              ** VRTC Kp trans-characteristics table index

* Kp trans-characteristics multiplier (and enable)

LD      xKpTransMul                ** Kp trans-characteristics table multiplier (<>0 == enable)
ST      VRTC_KP_TABLE_MUL          ** VRTC Kp trans-characteristics table multiplier

* Sliding mode deceleration

LD      xSlidingDecel
ST      VRTC_SLIDING_DECEL

LD      0
ST      VRTC_NON_LINEAR_MODE

LD      xSlidingDecel
EQ      0
JMPC    endif_non_linear_mode
    LD      1
    ST      VRTC_NON_LINEAR_MODE
endif_non_linear_mode:

LD      xKpTransMul                ** Kp trans-characteristics table multiplier (<>0 == enable)
NE      0
OR (
	LD      xSlidingDecel
	NE      0
)
ST      CtrReg0.17          * Enable Kp trans-characteristics

* Kp deadband

LD      xDbPos                     ** positive deadband
ST      VRTC_DB_POS                ** VRTC positive deadband
LD      xDbNeg                     ** negative deadband
ST      VRTC_DB_NEG                ** VRTC negative deadband

**** can be disabled by simply setting parameter to 0
LD      %PLCFLAGS.1
ST      CtrReg0.8           * Enable deadband processing

* Filter cutoff frequency

LD      xFilterCutOff              ** Filter cutoff frequency [Hz]
ST      VRTC_CUTOFF                ** VRTC Filter cutoff frequency [Hz]

* filter Damping

LD      xFilterDamping             ** Filter Damping Coefficient
ST      VRTC_DAMPING               ** VRTC Damping filter

* Error Fading Time

LD      xSimFadingTime             ** Simulation Xfade time [ms]
ST      VRTC_SIM_FADER             ** VRTC Simulation Xfade time [ms]

**** can be disabled by simply setting parameter to 0
LD      %PLCFLAGS.1
ST      CtrReg0.11          * Enable off-sensor simulation fader

* Velocity lock trigger (always enabled)

LD      xLockVelLimitUp            ** Lock trigger velocity Up
ST      VRTC_TRIG_VEL_UP           ** VRTC Lock trigger velocity Up
LD      xLockVelLimitDown          ** Lock trigger velocity Down
ST      VRTC_TRIG_VEL_LW           ** VRTC Lock trigger velocity Down

LD      %PLCFLAGS.1
ST      CtrReg1.16                  * Enable velocity lock trigger

* Acceleration lock trigger (enabled if <> 0)

LD      xLockAccLimit              ** Lock trigger acceleration
ST      VRTC_TRIG_ACC              ** VRTC Lock trigger acceleration

LD      xLockAccLimit              ** Lock trigger acceleration
NE      0
ST      CtrReg1.17                  * Enable acceleration lock trigger

* ***

LD      xMLonlyClampFilterIn
ST      CtrReg1.11

LD      xMLonlyClampFilterInDot
ST      CtrReg1.10

* Simulation offset set

LDN   xReset                ** Reset
JMPC  not_reset

    LD   0
    ST   VRTC_SIM_OFFSET_SET    ** VRTC simulation offset set

    JMP  endif_offset
not_reset:

LD   xSimul                        ** Simulazione
ORN  VRTC_SR0.28                   * VSR0_SIM_FADED_OUT
    JMPC simul

    LD   VRTC_SIM_OFFSET_CUR        ** VRTC simulation offset cur
    ST   VRTC_SIM_OFFSET_SET        ** VRTC simulation offset set

    JMP  endif_offset
simul:

    LDN  xMoveToTarget              ** Richiesta movimento su target
        JMPC endif_offset

        LD   xSimOffsetSet              ** VRTC simulation offset set
        ST   VRTC_SIM_OFFSET_SET        ** VRTC simulation offset set

endif_offset:

* Setpoint

LD   xSetPoint                     ** VRTC set point
ST   VRTC_SETPOINT                 ** VRTC setpoint

* Sensor input (commentare se non lo legge direttamente)

*** LD   xSensorIn           ** Sensor Input
*** ST   VRTC_SENSOR_IN      ** VRTC Sensor Input

* Trasferimento dati

CAL  TR_VRTSIM(CLK=xSimul)         ** Simulazione
CAL  TR_VRTRST(CLK=xReset)         ** Reset
CAL  TR_VRTRPI(CLK=xResPosInt)     ** Reset position integrator
CAL  TR_VRTPLD(CLK=xPosLimDisab)   ** Disable mandatory position limit
CAL  TR_DEOVER(CLK=xDeOverlapEnab) ** Enable de-overlap
CAL  TR_ERRAMP(CLK=xErrorAmpEnab)  ** Enable error amplifier
CAL  TR_MLonlyClamp(CLK=xMLonlyClampFilterIn)
CAL  TR_MLonlyClampDot(CLK=xMLonlyClampFilterInDot)

LD   VRTC_SIM_OFFSET_SET           ** VRTC simulation offset set
NE   PrevSimOffsetSet              ** Valore precedente simulation offset set
AND  xSimul                        ** Simulazione
OR   (
LD   xUpPosLimit                   ** Mandatory upper position limit
NE   PrevUpPosLim                  ** Valore precedente mandatory upper position limit
)
OR   (
LD   xLwPosLimit                   ** Mandatory lower position limit
NE   PrevLwPosLim                  ** Valore precedente mandatory lower position limit
)
OR   (
LD   xVelLimitUp                   ** Upward Mandatory velocity limit
NE   PrevUpVelLim                  ** Valore precedente Up mandatory velocity limit
)
OR   (
LD   xVelLimitDown                 ** Downward Mandatory velocity limit
NE   PrevDnVelLim                  ** Valore precedente Down mandatory velocity limit
)
OR   (
LD   xAccLimitUp                   ** Upward Mandatory velocity limit
NE   PrevUpAccLim                  ** Valore precedente Up mandatory acceleration limi
)
OR   (
LD   xAccLimitDown                 ** Downward Mandatory velocity limit
NE   PrevDnAccLim                  ** Valore precedente Down mandatory acceleration limit
)
OR(
LD   xKpGain                       ** Kp gain [[mm/s]/U]
NE   PrevKpGain                    ** Valore precedente Kp gain
)
OR   (
LD   xKpTransPtr                   ** Kp trans-characteristics table index
NE   PrevKpTransPtr                ** Previous Kp trans-characteristics table index
)
OR   (
LD   xKpTransMul                   ** Kp trans-characteristics table multiplier (<>0 == enable)
NE   PrevKpTransMul                ** Previous Kp trans-characteristics table multiplier (<>0 == enable)
)
OR(
LD   xSlidingDecel
NE   PrevSlidingDecel
)
OR   (
LD   xDbPos                        ** positive deadband
NE   PrevDbPos                     ** Previous positive deadband
)
OR   (
LD   xDbNeg                        ** negative deadband
NE   PrevDbNeg                     ** Previous negative deadband
)
OR(
LD   xFilterCutOff                 ** Filter cutoff frequency [Hz]
NE   PrevFilterCutOff              ** Previous Filter cutoff frequency
)
OR(
LD   xFilterDamping                ** Filter Damping Coefficient
NE   PrevFilterDamping             ** Previous filter damping value
)
OR   (
LD   xSimFadingTime                ** Simulation Xfade time [ms]
NE   PrevSimFadingTime             ** Previous Simulation Xfade time [ms]
)
OR   (
LD   xLockVelLimitUp               ** Lock trigger velocity Up
NE   PrevLockVelLimitUp            ** Previous Lock trigger velocity Up
)
OR   (
LD   xLockVelLimitDown             ** Lock trigger velocity Down
NE   PrevLockVelLimitDn            ** Previous Lock trigger velocity Down
)
OR   (
LD   xLockAccLimit                 ** Lock trigger acceleration
NE   PrevLockAccLimit              ** Previous Lock trigger acceleration
)
OR   (
LD   xSetPoint                     ** Setpoint
NE   PrevSetpoint                  ** Previous setpoint
)
OR   TR_MLonlyClamp.Q
OR   TR_MLonlyClampDot.Q
OR   TR_VRTSIM.Q                   ** Simulazione
OR   TR_VRTRST.Q                   ** Reset VRTC
OR   TR_VRTRPI.Q                   ** Imp. reset position integrator
OR   TR_VRTPLD.Q                   ** Imp. disable mandatory position limit
OR   TR_DEOVER.Q                   ** Enable de-overlap
OR   TR_ERRAMP.Q                   ** Enable error amplifier
JMPCN END_T_VRTCMD

LDN  CtrReg0.28          * Toggle bit #0
ST   CtrReg0.28          * Toggle bit #0

END_T_VRTCMD:

LD   VRTC_SIM_OFFSET_SET           ** VRTC simulation offset set
ST   PrevSimOffsetSet              ** Valore precedente simulation offset set

LD   xUpPosLimit                   ** Mandatory upper position limit
ST   PrevUpPosLim                  ** Valore precedente mandatory upper position limit

LD   xLwPosLimit                   ** Mandatory lower position limit
ST   PrevLwPosLim                  ** Valore precedente mandatory lower position limit

LD   xVelLimitUp                   ** Upward Mandatory velocity limit
ST   PrevUpVelLim                  ** Valore precedente Up mandatory velocity limit

LD   xVelLimitDown                 ** Downward Mandatory velocity limit
ST   PrevDnVelLim                  ** Valore precedente Down mandatory velocity limit

LD   xAccLimitUp                   ** Upward Mandatory velocity limit
ST   PrevUpAccLim                  ** Valore precedente Up mandatory acceleration limi

LD   xAccLimitDown                 ** Downward Mandatory velocity limit
ST   PrevDnAccLim                  ** Valore precedente Down mandatory acceleration limit

LD   xKpGain                       ** Kp gain [[mm/s]/U]
ST   PrevKpGain                    ** Valore precedente Kp gain

LD   xKpTransPtr                   ** Kp trans-characteristics table index
ST   PrevKpTransPtr                ** Previous Kp trans-characteristics table index

LD   xKpTransMul                   ** Kp trans-characteristics table multiplier (<>0 == enable)
ST   PrevKpTransMul                ** Previous Kp trans-characteristics table multiplier (<>0 == enable)

LD   xSlidingDecel
ST   PrevSlidingDecel

LD   xDbPos                        ** positive deadband
ST   PrevDbPos                     ** Previous positive deadband

LD   xDbNeg                        ** negative deadband
ST   PrevDbNeg                     ** Previous negative deadband

LD   xFilterCutOff                 ** Filter cutoff frequency [Hz]
ST   PrevFilterCutOff              ** Previous Filter cutoff frequency

LD   xFilterDamping                ** Filter Damping Coefficient
ST   PrevFilterDamping             ** Previous filter damping value

LD   xSimFadingTime                ** Simulation Xfade time [ms]
ST   PrevSimFadingTime             ** Previous Simulation Xfade time [ms]

LD   xLockVelLimitUp               ** Lock trigger velocity Up
ST   PrevLockVelLimitUp            ** Previous Lock trigger velocity Up

LD   xLockVelLimitDown             ** Lock trigger velocity Down
ST   PrevLockVelLimitDn            ** Previous Lock trigger velocity Down

LD   xLockAccLimit                 ** Lock trigger acceleration
ST   PrevLockAccLimit              ** Previous Lock trigger acceleration

LD   xSetPoint                     ** Setpoint
ST   PrevSetpoint                  ** Previous setpoint

LDN  CtrReg0.28          * Toggle bit #0
ST   CtrReg0.29          * Toggle bit #1

LD   CtrReg0.28          * Toggle bit #0
XOR  AckReg0.28          * Toggle strobe VRTC
ST   yBusy                         ** Comando VRTC in corso

LD   VRTC_SR0.8          * VSR0_SIGNAL_LOCK
ANDN yBusy                         ** Comando VRTC in corso
ANDN (
    LD   xSimul                         ** Simulazione
    ANDN VRTC_SR0.27                    * VSR0_SIM_FADED_IN
)
ANDN (
    LDN  xSimul                         ** Simulazione
    ANDN VRTC_SR0.28                    * VSR0_SIM_FADED_OUT
)
ANDN (
    LD   xErrorAmpEnab                  ** Enable error amplifier
    ANDN VRTC_SR0.25                    * VSR0_ERR_FADED_IN
)
ST   ySignalLock                   ** VRTC posizione raggiunta

LD   VRTC_SIM_OFFSET_CUR
ST   ySimOffsetCur

LD   VRTC_FLT_Q
ST   yFltQ

LD   CtrReg1                       ** Appoggio control register 1
ST   VRTC_CR1                      ** VRTC control register 1

LD   CtrReg0                       ** Appoggio control register 0
ST   VRTC_CR0                      ** VRTC control register 0

END_VRTC:

END_FUNCTION_BLOCK

FUNCTION_BLOCK GSTFEED

VAR_INPUT
ENC: WORD; * Quota da encoder (0-65535)
MUL: DWORD; * Moltiplicatore
MAXINC: DWORD; * Massimo incremento
END_VAR

VAR_OUTPUT
VAL: WORD; * Feedrate (0-120)
END_VAR

VAR
Multiplier:  DWORD;  *  Encoder feed multiplier
DiffQtaVolant: DWORD; * Differenza quota volantino rispetto alla precedente
QtaVolantAct: DWORD; * Quota volantino attuale
QtaVolantPrec: DWORD; * Quota volantino precedente
RETAIN FeedAx: DWORD; * Feedrate assi
END_VAR

* Carica la quota del volantino e fa la differenza con quella precedente

LD   ENC                           ** Quota da encoder (0-65535)
ST   QtaVolantAct                  ** Quota volantino attuale

LD   QtaVolantAct                  ** Quota volantino attuale
SUB  QtaVolantPrec                 ** Quota volantino precedente
ST   DiffQtaVolant                 ** Differenza quota volantino rispetto alla precedente

LD   QtaVolantAct                  ** Quota volantino attuale
ST   QtaVolantPrec                 ** Quota volantino precedente

* Estensione del segno da 16 a 32 bit

LD   DiffQtaVolant.15
JMPC SIGNEXT_NEGATIVE

LD   DiffQtaVolant                 ** Differenza quota volantino rispetto alla precedente
AND  16#0000FFFF
ST   DiffQtaVolant                 ** Differenza quota volantino rispetto alla precedente

LD   DiffQtaVolant                 ** Differenza quota volantino rispetto alla precedente
GT   MAXINC                        ** Massimo incremento
JMPCN LSF

LD   0
ST   DiffQtaVolant                 ** Differenza quota volantino rispetto alla precedente

LSF:

JMP  END_SIGNEXT

SIGNEXT_NEGATIVE:

LD   DiffQtaVolant                 ** Differenza quota volantino rispetto alla precedente
OR   16#FFFF0000
ST   DiffQtaVolant                 ** Differenza quota volantino rispetto alla precedente

END_SIGNEXT:

LDN   HW_ENCTYPE                   ** HW Type :0=S500, 1=S510
JMPC  S500
*S510:
LD   20
ST   Multiplier                    ** Encoder feed multiplier

JMP  END_S5X0

S500:

*LD   80
*LD   27

LD   MUL                           ** Moltiplicatore
ST   Multiplier                    ** Encoder feed multiplier
END_S5X0:

LD   DiffQtaVolant                 ** Differenza quota volantino rispetto alla precedente
MUL  Multiplier                    ** Moltiplicatore
ADD  FeedAx                        ** Feedrate assi
ST   FeedAx                        ** Feedrate assi

LD   FeedAx                        ** Feedrate assi
LT   0
JMPCN LFDN

LD   0
ST   FeedAx                        ** Feedrate assi

LFDN:

LD   FeedAx                        ** Feedrate assi
GT   4093
JMPCN LFUP

LD   4093
ST   FeedAx                        ** Feedrate assi

LFUP:

LD   FeedAx                        ** Feedrate assi
ST   VAL                           ** Feedrate (0-120)

END_FUNCTION_BLOCK
